# B&R Automation Studio project NAEUL004C00R13L518F00 (part 62)

#### Local.var
```iecst
(*2020-09-10*)
(**)
(*Local Action, State & Status*)
VAR
	eAct : eHermesAction := HermesActIdle;
	eStat : eHermesAction := HermesActIdle;
	eMainStatus : eFBStatus := Idle;
	eStatus : eFBStatus := Idle;
	eStatus1 : eFBStatus := Idle;
	eStatus2 : eFBStatus := Idle;
	eStatus3 : eFBStatus := Idle;
	eStatus4 : eFBStatus := Idle;
	udiStatus : UDINT := 0;
	udiStatus1 : UDINT := 0;
	udiStatus2 : UDINT := 0;
	udiStatus3 : UDINT := 0;
	udiStatus4 : UDINT := 0;
	udiStatus5 : UDINT := 0;
	sStatTxt : STRING[200] := '';
	a_sStatText : ARRAY[0..50] OF STRING[200] := ['Idling','Background Starting Operations','Background Stopping Operations','Deleting Old Log File','Creating Directory','Writing Retain File','Reading Retain File','Saving Configuration',43('')];
END_VAR
(**)
(*Local Alarm*)
VAR
	tyAlmData : tyAlmDat;
	tyAlmData1 : tyAlmDat;
	tyAlmData2 : tyAlmDat;
	tyAlmData3 : tyAlmDat;
	tyAlmData4 : tyAlmDat;
	tyAlmData5 : tyAlmDat;
	tyInfoData : tyAlmDat;
	tyInfoData1 : tyAlmDat;
	tyInfoData2 : tyAlmDat;
	a_tyAlmText : ARRAY[10000..10199] OF tyAlmTxt := [(sAlmText:='Invalid Ident While Client Connecting',sRcyText:='Problem Occurred In The TCP/IP Connection. Check The Connection And Try To Reconnect.'),(sAlmText:='Setting Keep Alive Interval Time Error While Client Connecting',sRcyText:='Unable To Establish Connection Between Machine. Check For Setting And Resume Operation.'),(sAlmText:='Setting Keep Alive Idle Time Error While Client Connecting',sRcyText:='Unable To Establish Connection Between Machine. Check For Setting And Resume Operation.'),(sAlmText:='Setting Keep Alive Count Error While Client Connecting',sRcyText:='Unable To Establish Connection Between Machine. Check For Setting And Resume Operation.'),(sAlmText:='Setting Keep Alive Error While Client Connecting',sRcyText:='Unable To Establish Connection Between Machine. Check For Setting And Resume Operation.'),(sAlmText:='Setting Receive Buffer Error While Client Connecting',sRcyText:='Unable To Establish Connection Between Machine. Check For Setting And Resume Operation.'),(sAlmText:='Setting Send Buffer Error While Client Connecting',sRcyText:='Unable To Establish Connection Between Machine. Check For Setting And Resume Operation.'),(sAlmText:='Setting No Waiting Error While Client Connecting',sRcyText:='Unable To Establish Connection Between Machine. Check For Setting And Resume Operation.'),(sAlmText:='TCP Open Port Error While Client Connecting',sRcyText:='Problem Occurred In The TCP/IP Connection. Check The Connection And Try To Reconnect.'),(sAlmText:='Closing TCP Error While Client Connecting',sRcyText:='Problem Occurred In The TCP/IP Connection. Check The Connection And Try To Reconnect.'),(sAlmText:='Server Connection Failed While Client Connecting',sRcyText:='There Was A Problem Connecting To The Server. The Server May Not Exist or It is Unavailable At This Time. Check The Connection and Try Again.'),(sAlmText:='Ident In Used While Client Connecting',sRcyText:='Problem Occurred In The TCP/IP Connection. Check The Connection And Reconnect.'),(sAlmText:='Connect To Server Error While Client Connecting',sRcyText:='There Was A Problem Connecting To The Server. The Server May Not Exist or It is Unavailable At This Time. Check The Connection and Try Again.'),(sAlmText:='US Hermes Connection Lost',sRcyText:='Please Check Network Connection.'),(sAlmText:='Invalid Ident While Receiving Data',sRcyText:='Problem Occurred In The TCP/IP Connection. Check The Connection And Try To Reconnect.'),(sAlmText:='TCP Receive Data Error While Receiving Data',sRcyText:='Problem Occurred In The TCP/IP Connection. Check The Connection And Try To Reconnect.'),(sAlmText:='Receive ServiceDescription While Upstream In Not Connected State',sRcyText:='Receive Illegal Message.'),(sAlmText:='Receive BoardAvailable While Upstream In Not Connected State',sRcyText:='Receive Illegal Message.'),(sAlmText:='Receive RevokeBoardAvailable While Upstream In Not Connected State',sRcyText:='Receive Illegal Message.'),(sAlmText:='Receive MachineReady While Upstream In Not Connected State',sRcyText:='Receive Illegal Message.'),(sAlmText:='Receive RevokeMachineReady While Upstream In Not Connected State',sRcyText:='Receive Illegal Message.'),(sAlmText:='Receive StartTransport While Upstream In Not Connected State',sRcyText:='Receive Illegal Message.'),(sAlmText:='Receive StopTransport While Upstream In Not Connected State',sRcyText:='Receive Illegal Message.'),(sAlmText:='Receive TransportFinished While Upstream In Not Connected State',sRcyText:='Receive Illegal Message.'),(sAlmText:='Receive BoardForecast While Upstream In Not Connected State',sRcyText:='Receive Illegal Message.'),(sAlmText:='Receive BoardAvailable While Upstream In Service Description State',sRcyText:='Receive Illegal Message.'),(sAlmText:='Receive RevokeBoardAvailable While Upstream In Service Description State',sRcyText:='Receive Illegal Message.'),(sAlmText:='Receive MachineReady While Upstream In Service Description State',sRcyText:='Receive Illegal Message.'),(sAlmText:='Receive RevokeMachineReady While Upstream In Service Description State',sRcyText:='Receive Illegal Message.'),(sAlmText:='Receive StartTransport While Upstream In Service Description State',sRcyText:='Receive Illegal Message.'),(sAlmText:='Receive StopTransport While Upstream In Service Description State',sRcyText:='Receive Illegal Message.'),(sAlmText:='Receive TransportFinished While Upstream In Service Description State',sRcyText:='Receive Illegal Message.'),(sAlmText:='Receive BoardForecast While Upstream In Service Description State',sRcyText:='Receive Illegal Message.'),(sAlmText:='Receive ServiceDescription While Upstream In Not Available Not Ready State',sRcyText:='Receive Illegal Message.'),(sAlmText:='Receive RevokeBoardAvailable While Upstream In Not Available Not Ready State',sRcyText:='Receive Illegal Message.'),(sAlmText:='Receive MachineReady While Upstream In Not Available Not Ready State',sRcyText:='Receive Illegal Message.'),(sAlmText:='Receive RevokeMachineReady While Upstream In Not Available Not Ready State',sRcyText:='Receive Illegal Message.'),(sAlmText:='Receive StartTransport While Upstream In Not Available Not Ready State',sRcyText:='Receive Illegal Message.'),(sAlmText:='Receive StopTransport While Upstream In Not Available Not Ready State',sRcyText:='Receive Illegal Message.'),(sAlmText:='Receive TransportFinished While Upstream In Not Available Not Ready State',sRcyText:='Receive Illegal Message.'),(sAlmText:='Receive ServiceDescription While Upstream In Board Available State',sRcyText:='Receive Illegal Message.'),(sAlmText:='Receive BoardAvailable While Upstream In Board Available State',sRcyText:='Receive Illegal Message.'),(sAlmText:='Receive MachineReady While Upstream In Board Available State',sRcyText:='Receive Illegal Message.'),(sAlmText:='Receive RevokeMachineReady While Upstream In Board Available State',sRcyText:='Receive Illegal Message.'),(sAlmText:='Receive StartTransport While Upstream In Board Available State',sRcyText:='Receive Illegal Message.'),(sAlmText:='Receive StopTransport While Upstream In Board Available State',sRcyText:='Receive Illegal Message.'),(sAlmText:='Receive TransportFinished While Upstream In Board Available State',sRcyText:='Receive Illegal Message.'),(sAlmText:='Receive BoardForecast While Upstream In Board Available State',sRcyText:='Receive Illegal Message.'),(sAlmText:='Receive ServiceDescription While Upstream In Machine Ready State',sRcyText:='Receive Illegal Message.'),(sAlmText:='Receive RevokeBoardAvailable While Upstream In Machine Ready State',sRcyText:='Receive Illegal Message.'),(sAlmText:='Receive MachineReady While Upstream In Machine Ready State',sRcyText:='Receive Illegal Message.'),(sAlmText:='Receive RevokeMachineReady While Upstream In Machine Ready State',sRcyText:='Receive Illegal Message.'),(sAlmText:='Receive StartTransport While Upstream In Machine Ready State',sRcyText:='Receive Illegal Message.'),(sAlmText:='Receive StopTransport While Upstream In Machine Ready State',sRcyText:='Receive Illegal Message.'),(sAlmText:='Receive TransportFinished While Upstream In Machine Ready State',sRcyText:='Receive Illegal Message.'),(sAlmText:='Receive ServiceDescription While Upstream In Available And Ready State',sRcyText:='Receive Illegal Message.'),(sAlmText:='Receive BoardAvailable While Upstream In Available And Ready State',sRcyText:='Receive Illegal Message.'),(sAlmText:='Receive MachineReady While Upstream In Available And Ready State',sRcyText:='Receive Illegal Message.'),(sAlmText:='Receive RevokeMachineReady While Upstream In Available And Ready State',sRcyText:='Receive Illegal Message.'),(sAlmText:='Receive StartTransport While Upstream In Available And Ready State',sRcyText:='Receive Illegal Message.'),(sAlmText:='Receive StopTransport While Upstream In Available And Ready State',sRcyText:='Receive Illegal Message.'),(sAlmText:='Receive TransportFinished While Upstream In Available And Ready State',sRcyText:='Receive Illegal Message.'),(sAlmText:='Receive BoardForecast While Upstream In Available And Ready State',sRcyText:='Receive Illegal Message.'),(sAlmText:='Receive ServiceDescription While Upstream In Transporting State',sRcyText:='Receive Illegal Message.'),(sAlmText:='Receive Twice Board Available While Upstream In Transporting State',sRcyText:='Receive Illegal Message.'),(sAlmText:='Receive RevokeBoardAvailable Without BoardAvailable While Upstream In Transporting State',sRcyText:='Receive Illegal Message.'),(sAlmText:='Receive MachineReady While Upstream In Transporting State',sRcyText:='Receive Illegal Message.'),(sAlmText:='Receive RevokeMachineReady While Upstream In Transporting State',sRcyText:='Receive Illegal Message.'),(sAlmText:='Receive StartTransport While Upstream In Transporting State',sRcyText:='Receive Illegal Message.'),(sAlmText:='Receive StopTransport While Upstream In Transporting State',sRcyText:='Receive Illegal Message.'),(sAlmText:='Receive ServiceDescription While Upstream In Transport Finished State',sRcyText:='Receive Illegal Message.'),(sAlmText:='Receive BoardAvailable While Upstream In Transport Finished State',sRcyText:='Receive Illegal Message.'),(sAlmText:='Receive RevokeBoardAvailable While UpstreamWhile Upstream In Transport Finished State',sRcyText:='Receive Illegal Message.'),(sAlmText:='Receive MachineReady While Upstream In Transport Finished State',sRcyText:='Receive Illegal Message.'),(sAlmText:='Receive RevokeMachineReady While Upstream In Transport Finished State',sRcyText:='Receive Illegal Message.'),(sAlmText:='Receive StartTransport While Upstream In Transport Finished State',sRcyText:='Receive Illegal Message.'),(sAlmText:='Receive TransportFinished While Upstream In Transport Finished State',sRcyText:='Receive Illegal Message.'),(sAlmText:='Receive StopTransport While Upstream In Transport Finished State',sRcyText:='Receive Illegal Message.'),(sAlmText:='Receive BoardForecast While Upstream In Transport Finished State',sRcyText:='Receive Illegal Message.'),(sAlmText:='Receive ServiceDescription While Upstream In Transport Stopped State',sRcyText:='Receive Illegal Message.'),(sAlmText:='Receive Twice Board Available While Upstream In Transport Stopped State',sRcyText:='Receive Illegal Message.'),(sAlmText:='Receive RevokeBoardAvailable Without BoardAvailable While Upstream In Transport Stopped State',sRcyText:='Receive Illegal Message.'),(sAlmText:='Receive MachineReady While Upstream In Transport Stopped State',sRcyText:='Receive Illegal Message.'),(sAlmText:='Receive RevokeMachineReady While Upstream In Transport Stopped State',sRcyText:='Receive Illegal Message.'),(sAlmText:='Receive StartTransport While Upstream In Transport Stopped State',sRcyText:='Receive Illegal Message.'),(sAlmText:='Receive StopTransport While Upstream In Transport Stopped State',sRcyText:='Receive Illegal Message.'),(sAlmText:='LaneId Mismatch While Checking Service Description',sRcyText:='The LaneId Value Does Not Match. Change The Value And Resend The Value.'),(sAlmText:='MachineId Missing While Checking Service Description',sRcyText:='Missing Input Value For MachineId. Fill Up The Value And Resend.'),(sAlmText:='LandId Out Of Range While Checking Service Description',sRcyText:='LaneId Does Not Fall Within The Expected Range.'),(sAlmText:='LandId Missing While Checking Service Description',sRcyText:='Missing Input Value For LaneId. Fill Up The Value And Resend.'),(sAlmText:='Version Missing While Checking Service Description',sRcyText:='Missing Input Value For Version. Fill Up The Value And Resend.'),(sAlmText:='SupportedFeatures Missing While Checking Service Description',sRcyText:='Missing Input Value For SupportedFeatures. Fill Up The Value And Resend.'),(sAlmText:='NotificationCode Out Of Range While Checking Notification',sRcyText:='NotificationCode Does Not Fall Within The Expected Range.'),(sAlmText:='NotificationCode Missing While Checking Notification',sRcyText:='Missing Input Value For NotificationCode. Fill Up The Value And Resend.'),(sAlmText:='Severity Missing While Checking Notification',sRcyText:='Missing Input Value For Severity. Fill Up The Value And Resend.'),(sAlmText:='Description Missing While Checking Notification',sRcyText:='Missing Input Value For Description. Fill Up The Value And Resend.'),(sAlmText:='BoardId Missing While Checking Board Available',sRcyText:='Missing Input Value For BoardId. Fill Up The Value And Resend.'),(sAlmText:='BoardIdCreatedBy Missing While Checking Board Available',sRcyText:='Missing Input Value For BoardIdCreatedBy. Fill Up The Value And Resend.'),(sAlmText:='FailedBoard Missing While Checking Board Available',sRcyText:='Missing Input Value For FailedBoard. Fill Up The Value And Resend.'),(sAlmText:='FlippedBoard Missing While Checking Board Available',sRcyText:='Missing Input Value For FlippedBoard. Fill Up The Value And Resend.'),(sAlmText:='TransferState Missing While Checking Transport Finished',sRcyText:='Missing Input Value For TransferState. Fill Up The Value And Resend.'),(sAlmText:='BoardId Missing While Checking Transport Finished',sRcyText:='Missing Input Value For BoardId. Fill Up The Value And Resend.'),(sAlmText:='FailedBoard Missing While Checking Board Forecast',sRcyText:='Missing Input Value For FailedBoard. Fill Up The Value And Resend.'),(sAlmText:='FlippedBoard Missing While Checking Board Forecast',sRcyText:='Missing Input Value For FlippedBoard. Fill Up The Value And Resend.'),(sAlmText:='BoardId Mismatch While Checking Start Transport & Transport Finished',sRcyText:='The BoardId Value Does Not Match. Change The Value And Resend The Value.'),(sAlmText:='BoardId Missing While Checking Start Transport & Transport Finished',sRcyText:='Missing Input Value For BoardId. Fill Up The Value And Resend.'),(sAlmText:='Service Description Interchange Time Out',sRcyText:='Timeout Expired Before Operation Completed. Reset And Resume Operation.'),(sAlmText:='Transport Time Out',sRcyText:='Timeout Expired Before Operation Completed. Reset And Resume Operation.'),(sAlmText:='Input First Slot Is Invalid',sRcyText:='Invalid Input Value.'),(sAlmText:='Input Last Slot Is Invalid',sRcyText:='Invalid Input Value.'),(sAlmText:='Input Pitch Is Invalid',sRcyText:='Invalid Input Value.'),(sAlmText:='Input Slot To Slot Distance Is Invalid',sRcyText:='Invalid Input Value.'),(sAlmText:='Input Total Slot Is Invalid',sRcyText:='Invalid Input Value.'),(sAlmText:='Input Thickness Is Invalid',sRcyText:='Invalid Input Value.'),(sAlmText:='Input Top Clearance Height Is Invalid',sRcyText:='Invalid Input Value.'),(sAlmText:='Input Bottom Clearance Height Is Invalid',sRcyText:='Invalid Input Value.'),(sAlmText:='Recipe First Slot Value & Board Available Data Not Match With Same Product Type Id',sRcyText:='The Recipe First Slot Value & Board Available Data Value Does Not Match With Product Type ID. Change The Value And Resend The Value.'),(sAlmText:='Recipe Last Slot Value & Board Available Data Not Match With Same Product Type Id',sRcyText:='The Recipe Last Slot Value & Board Available Data Value Does Not Match With Product Type ID. Change The Value And Resend The Value.'),(sAlmText:='Recipe Pitch Value & Board Available Data Not Match With Same Product Type Id',sRcyText:='The Recipe Pitch Value & Board Available Data Value Does Not Match With Product Type ID. Change The Value And Resend The Value.'),(sAlmText:='Width Different With Same Product Type Id',sRcyText:='Width Does Not Match With Product Type ID. Change The Value And Resend The Value.'),(sAlmText:='Input First Slot Is Invalid',sRcyText:='Invalid Input Value.'),(sAlmText:='Input Last Slot Is Invalid',sRcyText:='Invalid Input Value.'),(sAlmText:='Input Pitch Is Invalid',sRcyText:='Invalid Input Value.'),(sAlmText:='Input Slot To Slot Distance Is Invalid',sRcyText:='Invalid Input Value.'),(sAlmText:='Input Total Slot Is Invalid',sRcyText:='Invalid Input Value.'),(sAlmText:='Input Thickness Is Invalid',sRcyText:='Invalid Input Value.'),(sAlmText:='Input Top Clearance Height Is Invalid',sRcyText:='Invalid Input Value.'),(sAlmText:='Input Bottom Clearance Height Is Invalid',sRcyText:='Invalid Input Value.'),(sAlmText:='Recipe First Slot Value & Board Available Data Not Match With Same Product Type Id',sRcyText:='The Recipe First Slot Value & Board Available Data Value Does Not Match With Product Type ID. Change The Value And Resend The Value.'),(sAlmText:='Recipe Last Slot Value & Board Available Data Not Match With Same Product Type Id',sRcyText:='The Recipe Last Slot Value & Board Available Data Value Does Not Match With Product Type ID. Change The Value And Resend The Value.'),(sAlmText:='Recipe Pitch Value & Board Available Data Not Match With Same Product Type Id',sRcyText:='The Recipe Pitch Value & Board Available Data Value Does Not Match With Product Type ID. Change The Value And Resend The Value.'),(sAlmText:='Width Different With Same Product Type Id',sRcyText:='Width Does Not Match With Product Type ID. Change The Value And Resend The Value.'),(sAlmText:='Check Alive Time Out',sRcyText:='Timeout Expired Before Operation Completed. Reset And Resume Operation.'),(sAlmText:='Waiting Check Alive Time Out',sRcyText:='Timeout Expired Before Operation Completed. Reset And Resume Operation.'),(sAlmText:='Check Alive Id Mismatch',sRcyText:='The Check Alive Id Value Does Not Match. Change The Value And Resend The Value.'),(sAlmText:='Board Available Request To Send From Upstream Hermes',sRcyText:='Sending Illegal Message.'),(sAlmText:='Revoke Board Available Request To Send From Upstream Hermes',sRcyText:='Sending Illegal Message.'),(sAlmText:='Transport Finished Request To Send From Upstream Hermes',sRcyText:='Sending Illegal Message.'),(sAlmText:='Set Configuration Request To Send From Upstream Hermes',sRcyText:='Sending Illegal Message.'),(sAlmText:='Get Configuration Request To Send From Upstream Hermes',sRcyText:='Sending Illegal Message.'),(sAlmText:='Current Configuration Request To Send From Upstream Hermes',sRcyText:='Sending Illegal Message.'),(sAlmText:='Board Forecast Request To Send From Upstream Hermes',sRcyText:='Sending Illegal Message.'),(sAlmText:='Query Board Info Request To Send From Upstream Hermes',sRcyText:='Sending Illegal Message.'),(sAlmText:='Invalid Ident While Sending Data',sRcyText:='Invalid Ident Value.'),(sAlmText:='TCP Retry Send Data Error While Sending Data',sRcyText:='Problem Occurred In The TCP/IP Connection. Check The Connection And Try To Reconnect.'),(sAlmText:='TCP Send Data Error',sRcyText:='Problem Occurred In The TCP/IP Connection. Check The Connection And Try To Reconnect.'),(sAlmText:='Invalid Ident While Closing TCP',sRcyText:='Invalid Ident Value.'),(sAlmText:='Closing TCP Error',sRcyText:='Problem Occurred In The TCP/IP Connection. Check The Connection And Try To Reconnect.'),(sAlmText:='File Open Error While Writing Log',sRcyText:='An Error Was Encountered While Trying To Open File. Please Contact Nutek For A Possible Solution.'),(sAlmText:='File Create Error While Writing Log',sRcyText:='An Error Was Encountered While Trying To Create File. Please Contact Nutek For A Possible Solution.'),(sAlmText:='Get File Info Error While Writing Log',sRcyText:='An Error Was Encountered While Getting File Info. Please Contact Nutek For A Possible Solution.'),(sAlmText:='File Write Error While Writing Log',sRcyText:='An Error Was Encountered While Trying To Write File. Please Contact Nutek For A Possible Solution.'),(sAlmText:='File Close Error While Writing Log',sRcyText:='An Error Was Encountered While Trying To Close File. Please Contact Nutek For A Possible Solution.'),(sAlmText:='Directory Does Not Exist While Writing Log',sRcyText:='The Directory Does Not Exist.Please Contact Nutek For A Possible Solution.'),(sAlmText:='Get Directory Info Error While Deleting Old Log',sRcyText:='An Error Was Encountered While Getting Directory Info. Please Contact Nutek For A Possible Solution.'),(sAlmText:='Directory Read Error While Deleting Old Log',sRcyText:='An Error Was Encountered While Reading Directory. Please Contact Nutek For A Possible Solution.'),(sAlmText:='File Delete Error While Deleting Old Log',sRcyText:='An Error Was Encountered While Trying To Delete File. Please Contact Nutek For A Possible Solution.'),(sAlmText:='Board Jam At Sensor After Transfer Interrupted',sRcyText:='Push Back Board To Upstream Machine'),(sAlmText:='Product Type Id Not Receive From Upstream',sRcyText:='Check Upstream Machine Whether Product Type Id Is Used.'),(sAlmText:='Send Board Info Request To Send From Upstream Hermes',sRcyText:='Sending Illegal Message.'),(sAlmText:='Query Work Order Info Request To Send From Upstream Hermes',sRcyText:='Sending Illegal Message.'),(sAlmText:='Send Work Order Info Request To Send From Upstream Hermes',sRcyText:='Sending Illegal Message.'),(sAlmText:='Board Arrived Request To Send From Upstream Hermes',sRcyText:='Sending Illegal Message.'),(sAlmText:='Board Departed Request To Send From Upstream Hermes',sRcyText:='Sending Illegal Message.'),5((0)),(sAlmText:='New Recipe Not Found In Product Recipe List',sRcyText:='Create New Recipe In Product Setting.'),(sAlmText:='Top Barcode Mismatch While Checking SendBoardInfo & QueryBoardInfo',sRcyText:='Wrong Board Info Received. Pleae Check Again.'),(sAlmText:='Top Barcode Missing While Checking SendBoardInfo & QueryBoardInfo',sRcyText:='Wrong Board Info Received. Pleae Check Again.'),(sAlmText:='Bottom Barcode Mismatch While Checking SendBoardInfo & QueryBoardInfo',sRcyText:='Wrong Board Info Received. Pleae Check Again.'),(sAlmText:='Bottom Barcode Missing While Checking SendBoardInfo & QueryBoardInfo',sRcyText:='Wrong Board Info Received. Pleae Check Again.'),26((0))];
END_VAR
(**)
(*Local Output*)
VAR
	a_tyXMLTableDataBrdAvl : ARRAY[0..200] OF tyXMLTableDat;
	iXMLTableDataBrdAvlTtlIdx : INT;
	bConnected : BOOL;
	bHandshakeDone : BOOL;
	bAccDataReq : BOOL;
	bBFAccDataReq : BOOL;
	bOverWriteSlt : BOOL;
	bOverWriteWidth : BOOL;
	bBFOverWriteSlt : BOOL;
	bBFOverWriteWidth : BOOL;
	sReqRecipeNm : STRING[254];
	diReqWidthInUM : DINT;
	diReqMinSltValue : DINT;
	diReqMaxSltValue : DINT;
	diReqPitch : DINT;
	bNotAvlNotRdy : BOOL;
	bBoardAvailable : BOOL;
	bUSRdy : BOOL;
	bDSRdy : BOOL;
	bUSGdRdy : BOOL;
	bDSGdRdy : BOOL;
	bTransporting : BOOL;
	bStopTransport : BOOL;
	bBlkUS2 : BOOL;
	sInternalSnd : STRING[65535];
	bAccDataMnl : BOOL;
	bBFAccDataMnl : BOOL;
	bStopTransportSnd : BOOL;
	tyBoardArrivedInfo : tyHermesBoardAvailable;
	bRcvBoardInfoOk : BOOL;
	bRcvBoardInfoIncompl : BOOL;
	tySendBoardInfoAcc : tyHermesSendBoardInfo;
	tNextPCBTm : TIME;
	bBfReceivedInRdyState : BOOL;
	bBaReceivedInRdyState : BOOL;
END_VAR
(**)
(*Local Input*)
VAR
	udiRstErr : UDINT := 0;
	bPrep : BOOL := TRUE;
	bEn : BOOL := TRUE;
	bDis : BOOL := FALSE;
	tyParam : tyHermesUSParam := (tSndAlive:=T#30s,tRcvAlive:=T#60s,iLaneID:=1,sHostAddress:='192.168.0.200',uiHostPort:=5000);
	sIPAddr : STRING[15] := '192.168.0.100';
	tyDTStructure : DTStructure := (year:=2020,month:=11,day:=11,wday:=05,hour:=21,minute:=28,second:=30,millisec:=123,microsec:=456);
	dtCurrDT : DATE_AND_TIME := DT#2019-02-23-12:30:50;
	bRdyRcv : BOOL := FALSE;
	bRdyTransport : BOOL := FALSE;
	bRcvCompl : BOOL := FALSE;
	bRcvInCompl : BOOL := FALSE;
	bRcvNotStart : BOOL := FALSE;
	bBAWidthEn : BOOL := TRUE; (*Board Available Check Width*)
	bBASltEn : BOOL := FALSE; (*Board Available Check Slot*)
	bBFWidthEn : BOOL := TRUE; (*Board Forecast Check Width*)
	bBFSltEn : BOOL := FALSE; (*Board Forecast Check Slot*)
	sMcId : STRING[80] := '';
	sInterfaceId : STRING[80] := '';
	sVersion : STRING[7] := '1.3';
	eFailedBoard : eHermesFailedBoard := HermesUnknownBoard;
	sRecipeNm : STRING[254] := '';
	diWidthInUM : DINT := 0;
	diMinSltValue : DINT := 0;
	diMaxSltValue : DINT := 0;
	diPitch : DINT := 0;
	diTtlSlt : DINT := 0;
	diSltToSltInUM : DINT := 0;
	udiSndBffrSize : UDINT := 65536;
	udiRcvBffrSize : UDINT := 65536;
	udiAliveIdleTimeInSec : UDINT := 5;
	tConnTimeOut : TIME := T#30s;
	diTransferInTO : DINT := 30000;
	bOpsRun : BOOL := FALSE;
	bInterruptSen : BOOL := FALSE;
	udiFileKeepDay : UDINT := 30;
	sProgNm : STRING[15] := 'USHermes';
	bNtSettingsLoadDone : BOOL := TRUE;
	bAccDataRdy : BOOL := FALSE;
	bRmtPrep : BOOL := FALSE;
	bRmtEn : BOOL := FALSE;
	bSvyPrep : BOOL := FALSE;
	bSvyEn : BOOL := FALSE;
	bAccNewRcpCond : BOOL;
	sInfoMsg : STRING[200] := '';
	sInfoMsg1 : STRING[200] := '';
	sInfoMsg2 : STRING[200] := '';
	a_tyProdRcpList : ARRAY[1..c_udiProdRcpMax] OF tyProdRcpParam;
	tyProdRcpCurrRcp : tyProdRcpParam;
	bMcParamMnlAccData : BOOL;
	bUIAccData : BOOL;
	bQueryBoardInfo : BOOL;
	sTopBarcode : STRING[254] := '';
	sBottomBarcode : STRING[254] := '';
	bInternalUse : BOOL;
	sInternalRcv : STRING[65535];
	tyHermesCurrConfiguration : tyHermesConfiguration;
	bTransportFinished : BOOL;
	bManualInsertEndSen : BOOL;
	bManualInsertZoneHvBrd : BOOL;
	bOpsGConv1HvBrd : BOOL;
	bBAAccpt : BOOL;
	bBFAccpt : BOOL;
END_VAR
(**)
(*Local*)
VAR
	bRstErr : BOOL;
	udiRstErrOld : UDINT;
	bInitDone : BOOL;
	bInitialDone : BOOL;
	bRun : BOOL;
	bStop : BOOL;
	bRstConnection : BOOL;
	bRstState : BOOL;
	udiTCPIdent : UDINT;
	udiXMLTableWriteIdx : UDINT;
	udiMsgSendBffr : UDINT;
	udiSndMsgLen : UDINT;
	sSnd : STRING[65535];
	sRcv : STRING[65535];
	a_tyXMLTableDataRcv : ARRAY[0..200] OF tyXMLTableDat;
	a_tyXMLTableDataSnd : ARRAY[0..200] OF tyXMLTableDat;
	a_eMsgSend : ARRAY[0..50] OF eHermesMsgType;
	tyMsgTypeRcv : tyHermesMsgType;
	tyCheckAliveSnd : tyHermesCheckAlive;
	tyCheckAlivePingSnd : tyHermesCheckAlive;
	tyCheckAlivePongSnd : tyHermesCheckAlive;
	tyCheckAliveRcv : tyHermesCheckAlive;
	tyCheckAlivePingRcv : tyHermesCheckAlive;
	tyCheckAlivePongRcv : tyHermesCheckAlive;
	tyServiceDescriptionSnd : tyHermesServiceDescription;
	tyServiceDescriptionRcv : tyHermesServiceDescription;
	tyNotificationSnd : tyHermesNotification;
	tyNotificationRcv : tyHermesNotification;
	tyBoardAvailableRcv : tyHermesBoardAvailable;
	tyMachineReady : tyHermesMachineReady;
	tyStartTransport : tyHermesStartTransport;
	tyStopTransport : tyHermesStopTransport;
	tyTransportFinished : tyHermesTransportFinished;
	tySetConfiguration : tyHermesSetConfiguration;
	tyCurrentConfiguration : tyHermesCurrentConfiguration;
	tyBoardForecastAcc : tyHermesBoardForecast;
	tyBoardForecastRcv : tyHermesBoardForecast;
	tyQueryBoardInfo : tyHermesQueryBoardInfo;
	tySendBoardInfoRcv : tyHermesSendBoardInfo;
	fbClntConnect : fbTCPClntConnect;
	fbRcv : fbTCPRcv;
	fbSend : fbTCPSnd;
	fbClose : fbTCPClose;
	fbParseXMLTable : fbHermesParseXMLTable;
	fbCheckAlive : fbHermesCheckAlive;
	fbCheckAliveSendPing : fbHermesCheckAliveSendPing;
	fbCheckAliveRcvPing : fbHermesCheckAliveRcvPing;
	fbSequenceUS : fbHermesSequenceUS;
	fbSequenceTO : fbHermesSequenceTO;
	fbGetSlt : fbHermesGetSlt;
	eStatOld : eHermesAction := HermesActIdle;
	tyParamOld : tyHermesUSParam;
	bBlkUS : BOOL;
	bBABlkUS : BOOL;
	bBFBlkUS : BOOL;
	bManuallInsertLastZone : BOOL;
	udiLogCntr : UDINT := 1;
	udiWriteLogCntr : UDINT := 1;
	a_sLogList : ARRAY[1..10] OF STRING[65535];
	sDT : STRING[80];
	dtCurrDTTemp : DATE_AND_TIME;
	fbFileAppend1 : fbFileFullAppend;
	fbFileOldDel1 : fbFileOldDel;
	iWriteLogStep : INT := 0;
	i : INT;
	usiBFAccDataStep : USINT;
	usiAccDataStep : USINT;
	bFeatureBoardForecast : BOOL;
	bProcessBoardForecastId : BOOL;
	fbSendTm : TON;
	fbCheckBATimer : TON;
	fbDelayTm : TON;
	fbUSBlkTm : TON := (PT:=T#1s);
	bReplyMcRdyId : BOOL;
	fbDlyTmr : TON := (PT:=T#5s);
	fbDeleteLogTmr : TON := (PT:=T#24h);
	sTopBtmBarcode : ARRAY[0..1] OF STRING[254];
	udiModuleNum : UDINT := 3101;
END_VAR
```

#### Act_Alarm2.st
```iecst
(** 2019-03-25 **)
ACTION Act_Alarm2:

	//Error
	IF EDGEPOS(eStatus2 = Error) THEN

		tyAlmData2.sProgNm		:= p_sProgNm;
		tyAlmData2.udiCode		:= udiStatus2;
		tyAlmData2.eSeverity	:= AlmSeverityError;
		tyAlmData2.udiRunTime	:= tyAlmData2.udiRunTime + 1;
		tyAlmData2.bAlm			:= TRUE;
		tyAlmData2.udiModuleNum  := udiModuleNum;
		g_sUSHermesAProgNm		:= p_sProgNm;
		//Get Error Message
		IF tyAlmData2.udiCode < 10000 OR tyAlmData2.udiCode > 10199 THEN
			tyAlmData2.sAlmMsg	:= 'Unknown';
			tyAlmData2.sRcyMsg	:= 'Unknown';
		ELSE
			tyAlmData2.sAlmMsg	:= a_tyAlmText[tyAlmData2.udiCode].sAlmText;
			tyAlmData2.sRcyMsg	:= a_tyAlmText[tyAlmData2.udiCode].sRcyText;
		END_IF

		sStatTxt	:= tyAlmData2.sAlmMsg;

	ELSIF bRstErr AND (tyAlmData2.udiCode <> 0) THEN

		tyAlmData2.udiCode		:= 0;
		tyAlmData2.eSeverity	:= AlmSeverityNA;
		tyAlmData2.sAlmMsg		:= '';
		tyAlmData2.sRcyMsg		:= '';
		tyAlmData2.bAlm			:= FALSE;
		sStatTxt	:= a_sStatText[eStat];

	END_IF

END_ACTION
```

#### Act_Alarm4.st
```iecst
(** 2019-03-25 **)
ACTION Act_Alarm4:

	//Error
	IF EDGEPOS(eStatus4 = Error) THEN

		tyAlmData4.sProgNm		:= p_sProgNm;
		tyAlmData4.udiCode		:= udiStatus4;
		tyAlmData4.eSeverity	:= AlmSeverityError;
		tyAlmData4.udiRunTime	:= tyAlmData4.udiRunTime + 1;
		tyAlmData4.bAlm			:= TRUE;
		tyAlmData4.udiModuleNum  := udiModuleNum;
		g_sUSHermesAProgNm		:= p_sProgNm;
		//Get Error Message
		IF tyAlmData4.udiCode < 10000 OR tyAlmData4.udiCode > 10199 THEN
			tyAlmData4.sAlmMsg	:= 'Unknown';
			tyAlmData4.sRcyMsg	:= 'Unknown';
		ELSE
			tyAlmData4.sAlmMsg	:= a_tyAlmText[tyAlmData4.udiCode].sAlmText;
			tyAlmData4.sRcyMsg	:= a_tyAlmText[tyAlmData4.udiCode].sRcyText;
		END_IF

		sStatTxt	:= tyAlmData4.sAlmMsg;

	ELSIF bRstErr AND (tyAlmData4.udiCode <> 0) THEN

		tyAlmData4.udiCode		:= 0;
		tyAlmData4.eSeverity	:= AlmSeverityNA;
		tyAlmData4.sAlmMsg		:= '';
		tyAlmData4.sRcyMsg		:= '';
		tyAlmData4.bAlm			:= FALSE;
		sStatTxt	:= a_sStatText[eStat];

	END_IF

END_ACTION
```

#### Act_Alarm5.st
```iecst
(** 2020-09-10 **)
ACTION Act_Alarm5:

	//Error
	IF ((bConnected = FALSE) AND (p_eLinkMcParamUSCommMod= McSetCommModHermes)) THEN

		tyAlmData5.sProgNm		:= p_sProgNm;
		tyAlmData5.udiCode		:= udiStatus5;
		tyAlmData5.eSeverity	:= AlmSeverityWarning;
		tyAlmData5.udiRunTime	:= tyAlmData5.udiRunTime + 1;
		tyAlmData5.bWarning			:= TRUE;
		tyAlmData5.udiModuleNum  := udiModuleNum;
		g_sUSHermesAProgNm		:= p_sProgNm;
		//Get Error Message
		IF tyAlmData5.udiCode < 10000 OR tyAlmData5.udiCode > 10199 THEN
			tyAlmData5.sAlmMsg	:= 'Unknown';
			tyAlmData5.sRcyMsg	:= 'Unknown';
		ELSE
			tyAlmData5.sAlmMsg	:= a_tyAlmText[tyAlmData5.udiCode].sAlmText;
			tyAlmData5.sRcyMsg	:= a_tyAlmText[tyAlmData5.udiCode].sRcyText;
		END_IF

		sStatTxt	:= tyAlmData5.sAlmMsg;

	ELSIF (bConnected AND (tyAlmData5.udiCode <> 0)) OR (p_eLinkMcParamUSCommMod= McSetCommModSMEMA)  THEN

		tyAlmData5.udiCode		:= 0;
		tyAlmData5.eSeverity	:= AlmSeverityNA;
		tyAlmData5.sAlmMsg		:= '';
		tyAlmData5.sRcyMsg		:= '';
		tyAlmData5.bWarning			:= FALSE;
		sStatTxt	:= a_sStatText[eStat];

	END_IF

END_ACTION
```

#### Act_Background.st
```iecst
(** 2021-08-01 **)
ACTION Act_Background:

	IF bRun = TRUE THEN
		IF udiTCPIdent = 0 THEN
			IF p_bInternalUse = FALSE THEN
				Act_Background_TCPConnect;

				tyParamOld	:= p_tyParam;
			ELSE
				udiTCPIdent	:= 1;
			END_IF

		ELSE
			IF bRstConnection = FALSE THEN
				Act_Background_TCPRcv;

				Act_Background_NotificationRcv;
				Act_Background_IllegalMsg;
				Act_Background_ChkParamRcv;
				Act_Background_CmpParamRcv;

				IF bHandshakeDone = TRUE THEN
					IF (p_tyParam.tSndAlive <> T#0s) AND (p_tyParam.tRcvAlive <> T#0s) THEN
						IF tyServiceDescriptionRcv.tyData.tySupportedFeatures.bFeatureCheckAliveResponse = TRUE AND p_tyParam.bFeatureCheckAliveResponse = TRUE THEN
							Act_Background_ChkAliveSendPing;
							Act_Background_ChkAliveRcvPing;
						ELSE
							Act_Background_ChkAlive;
						END_IF
					ELSE
						fbCheckAlive(bEn := FALSE);
						fbCheckAliveSendPing(bEn := FALSE);
						fbCheckAliveRcvPing(bEn := FALSE);
					END_IF
				END_IF

				Act_Background_BoardAvailableChk;
				Act_Background_BoardForecastIdChk;
				Act_Background_Sequence;
				Act_Background_SequenceTO;
				Act_Background_Err;

				IF tyServiceDescriptionRcv.tyAvl.tySupportedFeatures.bFeatureSendBoardInfo = TRUE AND p_tyParam.bFeatureQueryBoardInfo AND bHandshakeDone THEN
					Act_Background_QueryBoardInfo;
				END_IF

				Act_Background_ChgConfig;

				Act_Background_TCPSend;

			//	Act_Background_Log;

			ELSE
				Act_Background_TCPClose;

			END_IF

		END_IF

	    Act_Background_Stop;

	END_IF
	Act_Background_Log;

	IF EDGENEG(bRun) OR EDGENEG(udiTCPIdent = 0) THEN
		//Reset
		fbClntConnect(bEn := FALSE);

		bConnected	:= bRun;
	END_IF

	IF EDGENEG(bRun) OR EDGENEG(udiTCPIdent <> 0) THEN
		fbRcv(bEn := FALSE);
		fbSequenceUS(bEn := FALSE);
		fbSequenceTO(bEn := FALSE);
		fbCheckAlive(bEn := FALSE);
		fbCheckAliveSendPing(bEn := FALSE);
		fbCheckAliveRcvPing(bEn := FALSE);
		fbSend(bEn := FALSE);
		fbClose(bEn := FALSE);

//		fbFileAppend1(bEn := FALSE);
//		iWriteLogStep	:= 0;

		bConnected		    := FALSE;
		bHandshakeDone	    := FALSE;
		bBlkUS			    := FALSE;
		bBABlkUS			:= FALSE;
		bBFBlkUS			:= FALSE;
		bManuallInsertLastZone	:= FALSE;
		bAccDataReq		    := FALSE;
		bBFAccDataReq	    := FALSE;
		bOverWriteSlt    	:= FALSE;
		bOverWriteWidth	    := FALSE;
		bBFOverWriteSlt	    := FALSE;
		bBFOverWriteWidth	:= FALSE;
		bRstConnection    	:= FALSE;
		bRstState	    	:= FALSE;
		bUSRdy	    		:= FALSE;
		bDSRdy		    	:= FALSE;
		bTransporting    	:= FALSE;
		bStopTransport   	:= FALSE;

		memset(ADR(tyMsgTypeRcv) , 0 , SIZEOF(tyMsgTypeRcv));
		memset(ADR(a_eMsgSend) , 0 , SIZEOF(a_eMsgSend));
		udiMsgSendBffr	:= 0;
	END_IF

	//Reset Error
	IF (eStatus1 = Error) AND bRstErr THEN
		eStatus1	:= Idle;
		udiStatus1	:= 0;

		fbClntConnect(bEn := FALSE);
		fbRcv(bEn := FALSE);
		fbSequenceUS(bEn := FALSE);
		fbSend(bEn := FALSE);
		fbClose(bEn := FALSE);
		fbCheckAlive(bEn := FALSE);
		fbCheckAliveSendPing(bEn := FALSE);
		fbCheckAliveRcvPing(bEn := FALSE);
		fbSequenceTO(bEn := FALSE);

//		fbFileAppend1(bEn := FALSE);
//		iWriteLogStep	:= 0;

		bConnected		    := FALSE;
		bHandshakeDone	    := FALSE;
		bBlkUS			    := FALSE;
		bBABlkUS			:= FALSE;
		bBFBlkUS			:= FALSE;
		bManuallInsertLastZone	:= FALSE;
		bAccDataReq		    := FALSE;
		bBFAccDataReq	    := FALSE;
		bOverWriteSlt    	:= FALSE;
		bOverWriteWidth	    := FALSE;
		bBFOverWriteSlt	    := FALSE;
		bBFOverWriteWidth	:= FALSE;
		bRstConnection    	:= FALSE;
		bRstState	    	:= FALSE;
		bUSRdy	    		:= FALSE;
		bDSRdy		    	:= FALSE;
		bTransporting    	:= FALSE;
		bStopTransport   	:= FALSE;

		memset(ADR(tyMsgTypeRcv) , 0 , SIZEOF(tyMsgTypeRcv));
		memset(ADR(a_eMsgSend) , 0 , SIZEOF(a_eMsgSend));
		udiMsgSendBffr	:= 0;
	END_IF

	IF (eStatus2 = Error) AND bRstErr THEN
		eStatus2	:= Idle;
		udiStatus2	:= 0;

		fbSequenceTO(bEn := FALSE);

	END_IF

	IF (eStatus3 = Error) AND bRstErr THEN
		eStatus3	:= Idle;
		udiStatus3	:= 0;

//		fbFileAppend1(bEn := FALSE);
//		iWriteLogStep	:= 0;
	END_IF

	IF (eStatus4 = Error) AND bRstErr THEN
		eStatus4	:= Idle;
		udiStatus4	:= 0;
	END_IF

	Act_Background_AccData;
	Act_Background_BFAccData;

END_ACTION
```

#### Act_Background_AccData.st
```iecst
(** 2021-08-01 **)
ACTION Act_Background_AccData: //Accept BoardAvailable Data from Upstream

	CASE usiAccDataStep OF
		0:
			//Request Accept Data
			IF bUSRdy = TRUE AND eMainStatus <> Error AND bAccDataReq = TRUE THEN
				usiAccDataStep	:= 1;
			END_IF
			//bUSRdy := fbSequenceUS.bUSRdy;
			//bUSRdy:= (eState = HermesStateBoardAvailable) OR (eState = HermesStateAvailableAndReady) OR (eState >= HermesStateTransporting);
		1:
			//Manual Accept Data Check
			IF bAccDataReq = TRUE THEN
				IF p_bMcParamMnlAccData = TRUE THEN
					bAccDataMnl	:= TRUE;

					tyInfoData.sProgNm		:= p_sProgNm;
					tyInfoData.udiCode		:= 10000;
					tyInfoData.eSeverity	:= AlmSeverityInfo;
					tyInfoData.sAlmMsg		:= p_sInfoMsg;

					IF p_bUIAccData = TRUE THEN
						p_bUIAccData    := FALSE; //2023_07_26_Debug for Manual Accept Data automatically accept after product change many times
						bAccDataMnl		:= FALSE;
						usiAccDataStep	:= 2;
					END_IF
				ELSE
					bAccDataMnl		:= FALSE;
					p_bUIAccData    := FALSE; //2023_07_26_Debug for Manual Accept Data automatically accept after product change many times
					usiAccDataStep	:= 2;
				END_IF
			ELSE
				bAccDataMnl		:= FALSE;
				usiAccDataStep	:= 4;
			END_IF

		2:
			IF bAccDataReq = TRUE  THEN
				IF p_bAccNewRcpCond = TRUE THEN //In Auto Mode, and empty
					usiAccDataStep	:= 3;
					IF p_bNtParamAutoRcpPrep AND NOT(p_bMcParamAutoRcpDis) THEN
						CASE p_eNtParamAutoRcpPrecededBy OF
							PrecededBySelf:
								usiAccDataStep	:= 4;
							PrecededByF1:
								usiAccDataStep	:= 3;
						END_CASE
					END_IF
				ELSE
					//Info Message
					tyInfoData.sProgNm		:= p_sProgNm;
					tyInfoData.udiCode		:= 10000;
					tyInfoData.eSeverity	:= AlmSeverityInfo;
					tyInfoData.sAlmMsg		:= p_sInfoMsg;
				END_IF
			ELSE
				usiAccDataStep	:= 4;
			END_IF

		3:
			//Sync Recipe
			IF bOverWriteWidth = TRUE OR bOverWriteSlt = TRUE THEN

				//Accept New Recipe Width
				IF bOverWriteWidth = TRUE THEN
					p_tyProdRcpCurrRcp.diWidthInUM	:= diReqWidthInUM;
				END_IF

				//Accept New Recipe Slot
				IF bOverWriteSlt = TRUE THEN
					p_tyProdRcpCurrRcp.diMaxSltValue := diReqMaxSltValue;
					p_tyProdRcpCurrRcp.diMinSltValue := diReqMinSltValue;
					p_tyProdRcpCurrRcp.diPitch		 := diReqPitch;
				END_IF

			ELSE

				//Accept New Recipe Name
				FOR i := 1 TO 2000 DO
					IF sReqRecipeNm = pa_tyProdRcpList[i].sRcpNm THEN
						p_tyProdRcpCurrRcp	:= pa_tyProdRcpList[i];
						EXIT;
					END_IF
				END_FOR

				IF i > 2000 THEN
					//Recipe Not Exist
					eStatus4	:= Error;
					udiStatus4	:= 10169;	//New Recipe Not Found In Product Recipe List

					fHermesAddOneMsgSend(ADR(a_eMsgSend) , ADR(udiMsgSendBffr) , HermesMsgTypeNotification);

					tyNotificationSnd.tyAvl.bSeverity			:= TRUE;
					tyNotificationSnd.tyAvl.bNotificationCode	:= TRUE;
					tyNotificationSnd.tyAvl.bDescription		:= TRUE;
					tyNotificationSnd.tyData.eSeverity			:= HermesSeverityError;
					tyNotificationSnd.tyData.iNotificationCode	:= UDINT_TO_INT(udiStatus4);
					tyNotificationSnd.tyData.sDescription		:= a_tyAlmText[udiStatus4].sAlmText;

				END_IF

			END_IF

			usiAccDataStep	:= 4;

		4:
			//Clear Info Message
			tyInfoData.sProgNm		:= '';
			tyInfoData.udiCode		:= 0;
			tyInfoData.eSeverity	:= AlmSeverityNA;
			tyInfoData.sAlmMsg		:= '';

			usiAccDataStep	:= 0;

	END_CASE

END_ACTION
```

#### Act_Background_BoardAvailableChk.st
```iecst
(** 2021-08-01 **)
ACTION Act_Background_BoardAvailableChk:

	IF eStatus2 <> Error THEN
		     //Add
		//IF p_bNewIncomingBoard = FALSE AND p_bSiemensMcModeChgPrep = FALSE AND
		IF p_bAccDataRdy AND (bTransporting = FALSE) AND(p_bOpsRun = TRUE) THEN
			bBaReceivedInRdyState	:= p_bAccDataRdy AND (bTransporting = FALSE) AND(p_bOpsRun = TRUE);//AutoRcp
			bAccDataReq		:= FALSE;
			bBABlkUS		:= FALSE;
			bOverWriteSlt	:= FALSE;
			bOverWriteWidth	:= FALSE;

			IF p_tyParam.bCmpTypeId = TRUE  THEN	//"Compare Type ID" Ticked

				IF tyBoardAvailableRcv.tyAvl.bProductTypeId = TRUE THEN	//Check if there is Product Type Id in B.A msg

					IF tyBoardAvailableRcv.tyData.sProductTypeId <> p_sRecipeNm THEN	//Product Type Id Different

						bAccDataReq	    := TRUE;	//Require To Load New Recipe
						bBABlkUS		:= TRUE;

						sReqRecipeNm	:= tyBoardAvailableRcv.tyData.sProductTypeId;
						diReqWidthInUM	:= REAL_TO_DINT(tyBoardAvailableRcv.tyData.rWidth * 1000);

					ELSE	//Product Type Id Same (After accepted or Originally same)

						IF p_tyParam.bCmpParam = TRUE THEN	//"Compare Param" Ticked
							IF tyBoardAvailableRcv.tyAvl.bThickness AND tyBoardAvailableRcv.tyAvl.bTopClearanceHeight AND tyBoardAvailableRcv.tyAvl.bBottomClearanceHeight AND p_bBASltEn THEN	//Camparing Slot Parameters if p_bBASltEn = TRUE
								udiStatus2	:= fHermesCmpSlt(tyBoardAvailableRcv.tyData.eFlippedBoard , tyBoardAvailableRcv.tyData.rThickness , tyBoardAvailableRcv.tyData.rTopClearanceHeight , tyBoardAvailableRcv.tyData.rBottomClearanceHeight , p_diMinSltValue , p_diMaxSltValue , p_diPitch , p_diSltToSltInUM , p_diTtlSlt);

								IF udiStatus2 <> 0 THEN

									bBABlkUS	:= TRUE;

									eStatus2	:= Error;

									IF udiStatus2 = 2914 THEN
										udiStatus2	:= 10108;	//Input First Slot Is Invalid
									ELSIF udiStatus2 = 2915 THEN
										udiStatus2	:= 10109;	//Input Last Slot Is Invalid
									ELSIF udiStatus2 = 2916 THEN
										udiStatus2	:= 10110;	//Input Pitch Is Invalid
									ELSIF udiStatus2 = 2917 THEN
										udiStatus2	:= 10111;	//Input Slot To Slot Distance Is Invalid
									ELSIF udiStatus2 = 2918 THEN
										udiStatus2	:= 10112;	//Input Total Slot Is Invalid
									ELSIF udiStatus2 = 2919 THEN
										udiStatus2	:= 10113;	//Input Thickness Is Invalid
									ELSIF udiStatus2 = 2920 THEN
										udiStatus2	:= 10114;	//Input Top Clearance Height Is Invalid
									ELSIF udiStatus2 = 2921 THEN
										udiStatus2	:= 10115;	//Input Bottom Clearance Height Is Invalid
									ELSIF udiStatus2 = 2922 THEN
										udiStatus2	:= 10116;	//Recipe First Slot Value & Board Available Data Not Match With Same Product Type Id
									ELSIF udiStatus2 = 2923 THEN
										udiStatus2	:= 10117;	//Recipe Last Slot Value & Board Available Data Not Match With Same Product Type Id
									ELSIF udiStatus2 = 2924 THEN
										udiStatus2	:= 10118;	//Recipe Pitch Value & Board Available Data Not Match With Same Product Type Id
									END_IF

									fHermesAddOneMsgSend(ADR(a_eMsgSend) , ADR(udiMsgSendBffr) , HermesMsgTypeNotification);

									tyNotificationSnd.tyAvl.bSeverity			:= TRUE;
									tyNotificationSnd.tyAvl.bNotificationCode	:= TRUE;
									tyNotificationSnd.tyAvl.bDescription		:= TRUE;
									tyNotificationSnd.tyData.eSeverity			:= HermesSeverityError;
									tyNotificationSnd.tyData.iNotificationCode	:= UDINT_TO_INT(udiStatus2);
									tyNotificationSnd.tyData.sDescription		:= a_tyAlmText[udiStatus2].sAlmText;

								END_IF
							END_IF

							IF tyBoardAvailableRcv.tyAvl.bWidth AND p_bBAWidthEn THEN	//Comparing Width Parameter if p_bBAWidthEn = TRUE
								IF REAL_TO_DINT(tyBoardAvailableRcv.tyData.rWidth * 1000) <> p_diWidthInUM THEN

									bBABlkUS	:= TRUE;

									eStatus2	:= Error;
									udiStatus2	:= 10119;	//Width Different With Same Product Type Id

									fHermesAddOneMsgSend(ADR(a_eMsgSend) , ADR(udiMsgSendBffr) , HermesMsgTypeNotification);

									tyNotificationSnd.tyAvl.bSeverity			:= TRUE;
									tyNotificationSnd.tyAvl.bNotificationCode	:= TRUE;
									tyNotificationSnd.tyAvl.bDescription		:= TRUE;
									tyNotificationSnd.tyData.eSeverity			:= HermesSeverityError;
									tyNotificationSnd.tyData.iNotificationCode	:= UDINT_TO_INT(udiStatus2);
									tyNotificationSnd.tyData.sDescription		:= a_tyAlmText[udiStatus2].sAlmText;

								END_IF
							END_IF

						END_IF

					END_IF

				ELSE

					eStatus2	:= Error;
					udiStatus2	:= 10158;	//Product Type Id Not Receive From Upstream

					fHermesAddOneMsgSend(ADR(a_eMsgSend) , ADR(udiMsgSendBffr) , HermesMsgTypeNotification);

					tyNotificationSnd.tyAvl.bSeverity			:= TRUE;
					tyNotificationSnd.tyAvl.bNotificationCode	:= TRUE;
					tyNotificationSnd.tyAvl.bDescription		:= TRUE;
					tyNotificationSnd.tyData.eSeverity			:= HermesSeverityError;
					tyNotificationSnd.tyData.iNotificationCode	:= UDINT_TO_INT(udiStatus2);
					tyNotificationSnd.tyData.sDescription		:= a_tyAlmText[udiStatus2].sAlmText;

				END_IF

			ELSE	//"Compare Type ID" Not Ticked
				                                    //Add
				IF p_tyParam.bOverwrite THEN //AND p_bNewIncomingBoard = FALSE  THEN	//"Overwrite" Ticked

					IF tyBoardAvailableRcv.tyAvl.bThickness AND tyBoardAvailableRcv.tyAvl.bTopClearanceHeight AND tyBoardAvailableRcv.tyAvl.bBottomClearanceHeight AND p_bBASltEn THEN	//Camparing Slot Parameters

						udiStatus2	:= fHermesCmpSlt(tyBoardAvailableRcv.tyData.eFlippedBoard , tyBoardAvailableRcv.tyData.rThickness , tyBoardAvailableRcv.tyData.rTopClearanceHeight , tyBoardAvailableRcv.tyData.rBottomClearanceHeight , p_diMinSltValue , p_diMaxSltValue , p_diPitch , p_diSltToSltInUM , p_diTtlSlt);

						IF udiStatus2 <> 0 THEN

							bAccDataReq		:= TRUE;
							bBABlkUS			:= TRUE;
							bOverWriteSlt	:= TRUE;

							fbGetSlt.eFlippedBrd				:= tyBoardAvailableRcv.tyData.eFlippedBoard;
							fbGetSlt.rThicknessInMM				:= tyBoardAvailableRcv.tyData.rThickness;
							fbGetSlt.rTopClearanceHeightInMM	:= tyBoardAvailableRcv.tyData.rTopClearanceHeight;
							fbGetSlt.rBtmClearanceHeightInMM	:= tyBoardAvailableRcv.tyData.rBottomClearanceHeight;
							fbGetSlt.diSltToSltInUM				:= p_diSltToSltInUM;
							fbGetSlt.diTtlSlt					:= p_diTtlSlt;
							fbGetSlt;

							diReqMinSltValue	:= fbGetSlt.diMinSltValue;
							diReqMaxSltValue	:= fbGetSlt.diMaxSltValue;
							diReqPitch			:= fbGetSlt.diPitch;

						END_IF

					END_IF

					IF tyBoardAvailableRcv.tyAvl.bWidth  AND p_bBAWidthEn THEN // AND p_usiLinkProdRcpCurrRcpMcMod = 0 THEN	//Comparing Width Parameter
						IF REAL_TO_DINT(tyBoardAvailableRcv.tyData.rWidth * 1000) <> p_diWidthInUM THEN

							bAccDataReq		:= TRUE;
							bBABlkUS		:= TRUE;
							bOverWriteWidth	:= TRUE;

							diReqWidthInUM	:= REAL_TO_DINT(tyBoardAvailableRcv.tyData.rWidth * 1000);

						END_IF
					END_IF

				ELSE	//"Compare Type ID" Not Ticked and "Overwrite" Not Ticked, Error if not same

					IF tyBoardAvailableRcv.tyAvl.bThickness AND tyBoardAvailableRcv.tyAvl.bTopClearanceHeight AND tyBoardAvailableRcv.tyAvl.bBottomClearanceHeight AND p_bBASltEn AND p_bRdyRcv THEN	//Camparing Slot Parameters
						udiStatus2	:= fHermesCmpSlt(tyBoardAvailableRcv.tyData.eFlippedBoard , tyBoardAvailableRcv.tyData.rThickness , tyBoardAvailableRcv.tyData.rTopClearanceHeight , tyBoardAvailableRcv.tyData.rBottomClearanceHeight , p_diMinSltValue , p_diMaxSltValue , p_diPitch , p_diSltToSltInUM , p_diTtlSlt);

						IF udiStatus2 <> 0 THEN

							bBABlkUS		:= TRUE;

							eStatus2	:= Error;

							IF udiStatus2 = 2914 THEN
								udiStatus2	:= 10120;	//Input First Slot Is Invalid
							ELSIF udiStatus2 = 2915 THEN
								udiStatus2	:= 10121;	//Input Last Slot Is Invalid
							ELSIF udiStatus2 = 2916 THEN
								udiStatus2	:= 10122;	//Input Pitch Is Invalid
							ELSIF udiStatus2 = 2917 THEN
								udiStatus2	:= 10123;	//Input Slot To Slot Distance Is Invalid
							ELSIF udiStatus2 = 2918 THEN
								udiStatus2	:= 10124;	//Input Total Slot Is Invalid
							ELSIF udiStatus2 = 2919 THEN
								udiStatus2	:= 10125;	//Input Thickness Is Invalid
							ELSIF udiStatus2 = 2920 THEN
								udiStatus2	:= 10126;	//Input Top Clearance Height Is Invalid
							ELSIF udiStatus2 = 2921 THEN
								udiStatus2	:= 10127;	//Input Bottom Clearance Height Is Invalid
							ELSIF udiStatus2 = 2922 THEN
								udiStatus2	:= 10128;	//Recipe First Slot Value & Board Available Data Not Match With Same Product Type Id
							ELSIF udiStatus2 = 2923 THEN
								udiStatus2	:= 10129;	//Recipe Last Slot Value & Board Available Data Not Match With Same Product Type Id
							ELSIF udiStatus2 = 2924 THEN
								udiStatus2	:= 10130;	//Recipe Pitch Value & Board Available Data Not Match With Same Product Type Id
							END_IF

							fHermesAddOneMsgSend(ADR(a_eMsgSend) , ADR(udiMsgSendBffr) , HermesMsgTypeNotification);

							tyNotificationSnd.tyAvl.bSeverity			:= TRUE;
							tyNotificationSnd.tyAvl.bNotificationCode	:= TRUE;
							tyNotificationSnd.tyAvl.bDescription		:= TRUE;
							tyNotificationSnd.tyData.eSeverity			:= HermesSeverityError;
							tyNotificationSnd.tyData.iNotificationCode	:= UDINT_TO_INT(udiStatus2);
							tyNotificationSnd.tyData.sDescription		:= a_tyAlmText[udiStatus2].sAlmText;

						END_IF
					END_IF

					IF tyBoardAvailableRcv.tyAvl.bWidth AND p_bBAWidthEn AND p_bRdyRcv THEN	//Comparing Width Parameter
						IF REAL_TO_DINT(tyBoardAvailableRcv.tyData.rWidth * 1000) <> p_diWidthInUM THEN

							bBABlkUS		:= TRUE;

							eStatus2	:= Error;
							udiStatus2	:= 10131;	//Width Different With Same Product Type Id

							fHermesAddOneMsgSend(ADR(a_eMsgSend) , ADR(udiMsgSendBffr) , HermesMsgTypeNotification);

							tyNotificationSnd.tyAvl.bSeverity			:= TRUE;
							tyNotificationSnd.tyAvl.bNotificationCode	:= TRUE;
							tyNotificationSnd.tyAvl.bDescription		:= TRUE;
							tyNotificationSnd.tyData.eSeverity			:= HermesSeverityError;
							tyNotificationSnd.tyData.iNotificationCode	:= UDINT_TO_INT(udiStatus2);
							tyNotificationSnd.tyData.sDescription		:= a_tyAlmText[udiStatus2].sAlmText;

						END_IF
					END_IF

				END_IF

			END_IF

		ELSIF (p_bAccDataRdy = FALSE) OR bTransporting = TRUE THEN
			bBaReceivedInRdyState	:= FALSE;//AutoRcp
			bAccDataReq		:= FALSE;
			bBABlkUS		:= FALSE;
			bOverWriteSlt	:= FALSE;
			bOverWriteWidth	:= FALSE;
			sTopBtmBarcode[0] := tyBoardAvailableRcv.tyData.sTopBarcode;
			sTopBtmBarcode[1] := tyBoardAvailableRcv.tyData.sBottomBarcode;

		END_IF

	ELSE

		bAccDataReq		:= FALSE;
		bBABlkUS		:= TRUE;
		bOverWriteSlt	:= FALSE;
		bOverWriteWidth	:= FALSE;
		sTopBtmBarcode[0] 	:= '';
		sTopBtmBarcode[1] 	:= '';

		bBaReceivedInRdyState := FALSE; //AutoRcp
	END_IF

END_ACTION
```

#### Act_Background_BoardForecastIdChk.st
```iecst
(** 2021-08-01 **)
ACTION Act_Background_BoardForecastIdChk:

	IF eStatus2 <> Error  THEN

		IF bProcessBoardForecastId AND bNotAvlNotRdy AND (bTransporting = FALSE) AND (p_bOpsRun = TRUE) AND p_bSiemensMcModeChgPrep = FALSE THEN
			bBfReceivedInRdyState := 	bProcessBoardForecastId AND bNotAvlNotRdy AND (bTransporting = FALSE) AND (p_bOpsRun = TRUE)  ;	 //AutoRcp
			bBFAccDataReq		:= FALSE;
			bBFBlkUS			:= FALSE;
			bBFOverWriteSlt  	:= FALSE;
			bBFOverWriteWidth	:= FALSE;
			                                      //Add
			IF p_tyParam.bCmpTypeId = TRUE THEN // AND p_bNewIncomingBoard = FALSE  THEN	//"Compare Type ID" Ticked

				IF tyBoardForecastAcc.tyAvl.bProductTypeId = TRUE THEN	//Check if there is Product Type Id in B.F msg

					IF tyBoardForecastAcc.tyData.sProductTypeId <> p_sRecipeNm THEN	//Product Type Id Different

						bBFAccDataReq	:= TRUE;	//Require To Load New Recipe
						bBFBlkUS		:= TRUE;

						sReqRecipeNm	:= tyBoardForecastAcc.tyData.sProductTypeId;
						diReqWidthInUM	:= REAL_TO_DINT(tyBoardForecastAcc.tyData.rWidth * 1000);

					ELSE	//Product Type Id Same (After accepted or Originally same)

						IF p_tyParam.bCmpParam = TRUE THEN	//"Compare Param" Ticked
							IF tyBoardForecastAcc.tyAvl.bThickness AND tyBoardForecastAcc.tyAvl.bTopClearanceHeight AND tyBoardForecastAcc.tyAvl.bBottomClearanceHeight AND p_bBFSltEn THEN	//Camparing Slot Parameters if p_bBFSltEn = TRUE
								udiStatus2	:= fHermesCmpSlt(tyBoardForecastAcc.tyData.eFlippedBoard , tyBoardForecastAcc.tyData.rThickness , tyBoardForecastAcc.tyData.rTopClearanceHeight , tyBoardForecastAcc.tyData.rBottomClearanceHeight , p_diMinSltValue , p_diMaxSltValue , p_diPitch , p_diSltToSltInUM , p_diTtlSlt);

								IF udiStatus2 <> 0 THEN

									bBFBlkUS		:= TRUE;
									bProcessBoardForecastId := FALSE;//add
									eStatus2	:= Error;

									IF udiStatus2 = 2914 THEN
										udiStatus2	:= 10108;	//Input First Slot Is Invalid
									ELSIF udiStatus2 = 2915 THEN
										udiStatus2	:= 10109;	//Input Last Slot Is Invalid
									ELSIF udiStatus2 = 2916 THEN
										udiStatus2	:= 10110;	//Input Pitch Is Invalid
									ELSIF udiStatus2 = 2917 THEN
										udiStatus2	:= 10111;	//Input Slot To Slot Distance Is Invalid
									ELSIF udiStatus2 = 2918 THEN
										udiStatus2	:= 10112;	//Input Total Slot Is Invalid
									ELSIF udiStatus2 = 2919 THEN
										udiStatus2	:= 10113;	//Input Thickness Is Invalid
									ELSIF udiStatus2 = 2920 THEN
										udiStatus2	:= 10114;	//Input Top Clearance Height Is Invalid
									ELSIF udiStatus2 = 2921 THEN
										udiStatus2	:= 10115;	//Input Bottom Clearance Height Is Invalid
									ELSIF udiStatus2 = 2922 THEN
										udiStatus2	:= 10116;	//Recipe First Slot Value & Board Available Data Not Match With Same Product Type Id
									ELSIF udiStatus2 = 2923 THEN
										udiStatus2	:= 10117;	//Recipe Last Slot Value & Board Available Data Not Match With Same Product Type Id
									ELSIF udiStatus2 = 2924 THEN
										udiStatus2	:= 10118;	//Recipe Pitch Value & Board Available Data Not Match With Same Product Type Id
									END_IF

									fHermesAddOneMsgSend(ADR(a_eMsgSend) , ADR(udiMsgSendBffr) , HermesMsgTypeNotification);

									tyNotificationSnd.tyAvl.bSeverity			:= TRUE;
									tyNotificationSnd.tyAvl.bNotificationCode	:= TRUE;
									tyNotificationSnd.tyAvl.bDescription		:= TRUE;
									tyNotificationSnd.tyData.eSeverity			:= HermesSeverityError;
									tyNotificationSnd.tyData.iNotificationCode	:= 6; //BoardForecast Error
									tyNotificationSnd.tyData.sDescription		:= a_tyAlmText[udiStatus2].sAlmText;

								END_IF
							END_IF

							IF tyBoardForecastAcc.tyAvl.bWidth AND p_bBFWidthEn THEN	//Comparing Width Parameter if p_bBFWidthEn = TRUE
								IF REAL_TO_DINT(tyBoardForecastAcc.tyData.rWidth * 1000) <> p_diWidthInUM THEN

									bBFBlkUS	:= TRUE;
									bProcessBoardForecastId := FALSE;//add
									eStatus2	:= Error;
									udiStatus2	:= 10119;	//Width Different With Same Product Type Id

									fHermesAddOneMsgSend(ADR(a_eMsgSend) , ADR(udiMsgSendBffr) , HermesMsgTypeNotification);

									tyNotificationSnd.tyAvl.bSeverity			:= TRUE;
									tyNotificationSnd.tyAvl.bNotificationCode	:= TRUE;
									tyNotificationSnd.tyAvl.bDescription		:= TRUE;
									tyNotificationSnd.tyData.eSeverity			:= HermesSeverityError;
									tyNotificationSnd.tyData.iNotificationCode	:= 6; //BoardForecast Error
									tyNotificationSnd.tyData.sDescription		:= a_tyAlmText[udiStatus2].sAlmText;
								ELSE
									bReplyMcRdyId           := TRUE; //add
									bProcessBoardForecastId := FALSE; //add
								END_IF
							END_IF

						END_IF

					END_IF

				ELSE

					eStatus2	:= Error;
					udiStatus2	:= 10158;	//Product Type Id Not Receive From Upstream
					bProcessBoardForecastId := FALSE;//add

					fHermesAddOneMsgSend(ADR(a_eMsgSend) , ADR(udiMsgSendBffr) , HermesMsgTypeNotification);

					tyNotificationSnd.tyAvl.bSeverity			:= TRUE;
					tyNotificationSnd.tyAvl.bNotificationCode	:= TRUE;
					tyNotificationSnd.tyAvl.bDescription		:= TRUE;
					tyNotificationSnd.tyData.eSeverity			:= HermesSeverityError;
					tyNotificationSnd.tyData.iNotificationCode	:= 6; //BoardForecast Error
					tyNotificationSnd.tyData.sDescription		:= a_tyAlmText[udiStatus2].sAlmText;

				END_IF

			ELSE	//"Compare Type ID" Not Ticked

				IF p_tyParam.bOverwrite THEN // AND p_bNewIncomingBoard = FALSE   THEN	//"Overwrite" Ticked

					IF tyBoardForecastAcc.tyAvl.bThickness AND tyBoardForecastAcc.tyAvl.bTopClearanceHeight AND tyBoardForecastAcc.tyAvl.bBottomClearanceHeight AND p_bBFSltEn THEN	//Camparing Slot Parameters

						udiStatus2	:= fHermesCmpSlt(tyBoardForecastAcc.tyData.eFlippedBoard , tyBoardForecastAcc.tyData.rThickness , tyBoardForecastAcc.tyData.rTopClearanceHeight , tyBoardForecastAcc.tyData.rBottomClearanceHeight , p_diMinSltValue , p_diMaxSltValue , p_diPitch , p_diSltToSltInUM , p_diTtlSlt);

						IF udiStatus2 <> 0 THEN

							bBFAccDataReq		:= TRUE;
							bBFBlkUS			:= TRUE;
							bBFOverWriteSlt	    := TRUE;

							fbGetSlt.eFlippedBrd				:= tyBoardForecastAcc.tyData.eFlippedBoard;
							fbGetSlt.rThicknessInMM				:= tyBoardForecastAcc.tyData.rThickness;
							fbGetSlt.rTopClearanceHeightInMM	:= tyBoardForecastAcc.tyData.rTopClearanceHeight;
							fbGetSlt.rBtmClearanceHeightInMM	:= tyBoardForecastAcc.tyData.rBottomClearanceHeight;
							fbGetSlt.diSltToSltInUM				:= p_diSltToSltInUM;
							fbGetSlt.diTtlSlt					:= p_diTtlSlt;
							fbGetSlt;

							diReqMinSltValue	:= fbGetSlt.diMinSltValue;
							diReqMaxSltValue	:= fbGetSlt.diMaxSltValue;
							diReqPitch			:= fbGetSlt.diPitch;

						END_IF

					END_IF

					IF tyBoardForecastAcc.tyAvl.bWidth AND p_bBFWidthEn THEN	//Comparing Width Parameter
						IF REAL_TO_DINT(tyBoardForecastAcc.tyData.rWidth * 1000) <> p_diWidthInUM THEN

							bBFAccDataReq		:= TRUE;
							bBFBlkUS			:= TRUE;
							bBFOverWriteWidth	:= TRUE;

							diReqWidthInUM	:= REAL_TO_DINT(tyBoardForecastAcc.tyData.rWidth * 1000);
						ELSE
							bReplyMcRdyId           := TRUE; //add
							bProcessBoardForecastId := FALSE; //add
						END_IF
					END_IF

				ELSE	//"Compare Type ID" Not Ticked and "Overwrite" Not Ticked, Error if not same

					IF tyBoardForecastAcc.tyAvl.bThickness AND tyBoardForecastAcc.tyAvl.bTopClearanceHeight AND tyBoardForecastAcc.tyAvl.bBottomClearanceHeight AND p_bBFSltEn AND p_bRdyRcv THEN	//Camparing Slot Parameters
						udiStatus2	:= fHermesCmpSlt(tyBoardForecastAcc.tyData.eFlippedBoard , tyBoardForecastAcc.tyData.rThickness , tyBoardForecastAcc.tyData.rTopClearanceHeight , tyBoardForecastAcc.tyData.rBottomClearanceHeight , p_diMinSltValue , p_diMaxSltValue , p_diPitch , p_diSltToSltInUM , p_diTtlSlt);

						IF udiStatus2 <> 0 THEN

							bBFBlkUS		:= TRUE;
							bProcessBoardForecastId := FALSE;//add
							eStatus2	:= Error;

							IF udiStatus2 = 2914 THEN
								udiStatus2	:= 10120;	//Input First Slot Is Invalid
							ELSIF udiStatus2 = 2915 THEN
								udiStatus2	:= 10121;	//Input Last Slot Is Invalid
							ELSIF udiStatus2 = 2916 THEN
								udiStatus2	:= 10122;	//Input Pitch Is Invalid
							ELSIF udiStatus2 = 2917 THEN
								udiStatus2	:= 10123;	//Input Slot To Slot Distance Is Invalid
							ELSIF udiStatus2 = 2918 THEN
								udiStatus2	:= 10124;	//Input Total Slot Is Invalid
							ELSIF udiStatus2 = 2919 THEN
								udiStatus2	:= 10125;	//Input Thickness Is Invalid
							ELSIF udiStatus2 = 2920 THEN
								udiStatus2	:= 10126;	//Input Top Clearance Height Is Invalid
							ELSIF udiStatus2 = 2921 THEN
								udiStatus2	:= 10127;	//Input Bottom Clearance Height Is Invalid
							ELSIF udiStatus2 = 2922 THEN
								udiStatus2	:= 10128;	//Recipe First Slot Value & Board Available Data Not Match With Same Product Type Id
							ELSIF udiStatus2 = 2923 THEN
								udiStatus2	:= 10129;	//Recipe Last Slot Value & Board Available Data Not Match With Same Product Type Id
							ELSIF udiStatus2 = 2924 THEN
								udiStatus2	:= 10130;	//Recipe Pitch Value & Board Available Data Not Match With Same Product Type Id
							END_IF

							fHermesAddOneMsgSend(ADR(a_eMsgSend) , ADR(udiMsgSendBffr) , HermesMsgTypeNotification);

							tyNotificationSnd.tyAvl.bSeverity			:= TRUE;
							tyNotificationSnd.tyAvl.bNotificationCode	:= TRUE;
							tyNotificationSnd.tyAvl.bDescription		:= TRUE;
							tyNotificationSnd.tyData.eSeverity			:= HermesSeverityError;
							tyNotificationSnd.tyData.iNotificationCode	:= 6; //BoardForecast Error
							tyNotificationSnd.tyData.sDescription		:= a_tyAlmText[udiStatus2].sAlmText;

						END_IF
					END_IF

					IF tyBoardForecastAcc.tyAvl.bWidth AND p_bBFWidthEn AND p_bRdyRcv THEN	//Comparing Width Parameter
						IF REAL_TO_DINT(tyBoardForecastAcc.tyData.rWidth * 1000) <> p_diWidthInUM THEN

							bBFBlkUS		:= TRUE;
							bProcessBoardForecastId := FALSE;//add
							eStatus2	:= Error;
							udiStatus2	:= 10131;	//Width Different With Same Product Type Id

							fHermesAddOneMsgSend(ADR(a_eMsgSend) , ADR(udiMsgSendBffr) , HermesMsgTypeNotification);

							tyNotificationSnd.tyAvl.bSeverity			:= TRUE;
							tyNotificationSnd.tyAvl.bNotificationCode	:= TRUE;
							tyNotificationSnd.tyAvl.bDescription		:= TRUE;
							tyNotificationSnd.tyData.eSeverity			:= HermesSeverityError;
							tyNotificationSnd.tyData.iNotificationCode	:= 6; //BoardForecast Error
							tyNotificationSnd.tyData.sDescription		:= a_tyAlmText[udiStatus2].sAlmText;
						ELSE
							bReplyMcRdyId           := TRUE; //add
							bProcessBoardForecastId := FALSE; //add
						END_IF
					END_IF

				END_IF

			END_IF

		ELSIF bProcessBoardForecastId = FALSE OR bNotAvlNotRdy =FALSE OR bTransporting = TRUE THEN
			bBfReceivedInRdyState := 	FALSE;
			bBFAccDataReq		:= FALSE;
			bBFBlkUS			:= FALSE;
			bBFOverWriteSlt	    := FALSE;
			bBFOverWriteWidth	:= FALSE;

		END_IF

	ELSE

		bBFAccDataReq		:= FALSE;
		bBFBlkUS			:= TRUE;
		bBFOverWriteSlt	    := FALSE;
		bBFOverWriteWidth	:= FALSE;

		bBfReceivedInRdyState := FALSE; //AutoRcp
	END_IF

END_ACTION
```

#### Act_Background_ChkAlive.st
```iecst
(** 2021-08-01 **)
ACTION Act_Background_ChkAlive:

	IF eStatus1 <> Error THEN

		//Standard Check Alive (Without Ping & Pong)
		fbCheckAlive.bDataRcv		:= tyMsgTypeRcv.bCheckAlive OR tyMsgTypeRcv.bBoardAvailable OR tyMsgTypeRcv.bRevokeBoardAvailable OR tyMsgTypeRcv.bTransportFinished OR tyMsgTypeRcv.bBoardForecast OR tyMsgTypeRcv.bSendBoardInfo;
		fbCheckAlive.tSendTm		:= p_tyParam.tSndAlive;
		fbCheckAlive.tRcvTimeOut	:= p_tyParam.tRcvAlive;
		fbCheckAlive(bEn := TRUE);

		IF fbCheckAlive.udiStatus > 0 AND fbCheckAlive.udiStatus < 65534 THEN
			eStatus1	:= Error;

			IF fbCheckAlive.udiStatus = 2767 THEN
				udiStatus1	:= 10132;	//Check Alive Time Out
			ELSE
				udiStatus1	:= fbCheckAlive.udiStatus;
			END_IF

			fHermesAddOneMsgSend(ADR(a_eMsgSend) , ADR(udiMsgSendBffr) , HermesMsgTypeNotification);

			tyNotificationSnd.tyAvl.bSeverity			:= TRUE;
			tyNotificationSnd.tyAvl.bNotificationCode	:= TRUE;
			tyNotificationSnd.tyAvl.bDescription		:= TRUE;
			tyNotificationSnd.tyData.eSeverity			:= HermesSeverityFatalError;
			tyNotificationSnd.tyData.iNotificationCode	:= UDINT_TO_INT(udiStatus1);
			tyNotificationSnd.tyData.sDescription		:= a_tyAlmText[udiStatus1].sAlmText;

		ELSE
			IF EDGEPOS(fbCheckAlive.bDataSend) THEN
				fHermesAddOneMsgSend(ADR(a_eMsgSend) , ADR(udiMsgSendBffr) , HermesMsgTypeCheckAlive);
				tyCheckAliveSnd	:= fbCheckAlive.tyDataSend;
			END_IF

		END_IF

		tyMsgTypeRcv.bCheckAlive	:= FALSE;	//Reset Check Alive

	END_IF

END_ACTION
```

#### Act_Background_ChkParamRcv.st
```iecst
(** 2021-08-01 **)
ACTION Act_Background_ChkParamRcv:

	IF eStatus2 <> Error THEN

		//Check Parameter Receive
		IF tyMsgTypeRcv.bServiceDescription = TRUE THEN
			udiStatus2	:= fHermesChkParamSD(tyServiceDescriptionRcv , p_tyParam.iLaneID);

			IF udiStatus2 = 2731 THEN
				udiStatus2	:= 0;
			END_IF

			IF udiStatus2 <> 0 THEN
				eStatus2	:= Error;

				IF udiStatus2 = 2726 THEN
					udiStatus2	:= 10086;	//LaneId Mismatch While Checking Service Description
				ELSIF udiStatus2 = 2727 THEN
					udiStatus2	:= 10087;	//MachineId Missing While Checking Service Description
				ELSIF udiStatus2 = 2728 THEN
					udiStatus2	:= 10088;	//LandId Out Of Range While Checking Service Description
				ELSIF udiStatus2 = 2729 THEN
					udiStatus2	:= 10089;	//LandId Missing While Checking Service Description
				ELSIF udiStatus2 = 2730 THEN
					udiStatus2	:= 10090;	//Version Missing While Checking Service Description
				ELSIF udiStatus2 = 2731 THEN
					udiStatus2	:= 10091;	//SupportedFeatures Missing While Checking Service Description
				END_IF

				fHermesAddOneMsgSend(ADR(a_eMsgSend) , ADR(udiMsgSendBffr) , HermesMsgTypeNotification);

				tyNotificationSnd.tyAvl.bSeverity			:= TRUE;
				tyNotificationSnd.tyAvl.bNotificationCode	:= TRUE;
				tyNotificationSnd.tyAvl.bDescription		:= TRUE;
				tyNotificationSnd.tyData.eSeverity			:= HermesSeverityFatalError;
				tyNotificationSnd.tyData.iNotificationCode	:= UDINT_TO_INT(udiStatus2);
				tyNotificationSnd.tyData.sDescription		:= a_tyAlmText[udiStatus2].sAlmText;

			END_IF
		END_IF

		IF tyMsgTypeRcv.bNotification = TRUE THEN
			udiStatus2	:= fHermesChkParamN(tyNotificationRcv);

			IF udiStatus2 <> 0 THEN
				eStatus2	:= Error;

				IF udiStatus2 = 2732 THEN
					udiStatus2	:= 10092;	//NotificationCode Out Of Range While Checking Notification
				ELSIF udiStatus2 = 2733 THEN
					udiStatus2	:= 10093;	//NotificationCode Missing While Checking Notification
				ELSIF udiStatus2 = 2734 THEN
					udiStatus2	:= 10094;	//Severity Missing While Checking Notification
				ELSIF udiStatus2 = 2735 THEN
					udiStatus2	:= 10095;	//Description Missing While Checking Notification
				END_IF

				fHermesAddOneMsgSend(ADR(a_eMsgSend) , ADR(udiMsgSendBffr) , HermesMsgTypeNotification);

				tyNotificationSnd.tyAvl.bSeverity			:= TRUE;
				tyNotificationSnd.tyAvl.bNotificationCode	:= TRUE;
				tyNotificationSnd.tyAvl.bDescription		:= TRUE;
				tyNotificationSnd.tyData.eSeverity			:= HermesSeverityFatalError;
				tyNotificationSnd.tyData.iNotificationCode	:= UDINT_TO_INT(udiStatus2);
				tyNotificationSnd.tyData.sDescription		:= a_tyAlmText[udiStatus2].sAlmText;

			END_IF
		END_IF

		IF tyMsgTypeRcv.bBoardAvailable = TRUE THEN
			udiStatus2	:= fHermesChkParamBA(tyBoardAvailableRcv);

			IF udiStatus2 <> 0 THEN
				eStatus2	:= Error;

				IF udiStatus2 = 2736 THEN
					udiStatus2	:= 10096;	//BoardId Missing While Checking Board Available
				ELSIF udiStatus2 = 2737 THEN
					udiStatus2	:= 10097;	//BoardIdCreatedBy Missing While Checking Board Available
				ELSIF udiStatus2 = 2738 THEN
					udiStatus2	:= 10098;	//FailedBoard Missing While Checking Board Available
				ELSIF udiStatus2 = 2739 THEN
					udiStatus2	:= 10099;	//FlippedBoard Missing While Checking Board Available
				END_IF

				fHermesAddOneMsgSend(ADR(a_eMsgSend) , ADR(udiMsgSendBffr) , HermesMsgTypeNotification);

				tyNotificationSnd.tyAvl.bSeverity			:= TRUE;
				tyNotificationSnd.tyAvl.bNotificationCode	:= TRUE;
				tyNotificationSnd.tyAvl.bDescription		:= TRUE;
				tyNotificationSnd.tyData.eSeverity			:= HermesSeverityError;
				tyNotificationSnd.tyData.iNotificationCode	:= UDINT_TO_INT(udiStatus2);
				tyNotificationSnd.tyData.sDescription		:= a_tyAlmText[udiStatus2].sAlmText;
//			ELSE
//				IF p_bNtParamAutoRcpPrep AND NOT(p_bMcParamAutoRcpDis) THEN
//					bBAAccpt := TRUE;
//				END_IF
			END_IF
//		ELSE
//			bBAAccpt := FALSE;
		END_IF

		IF tyMsgTypeRcv.bTransportFinished = TRUE THEN
			udiStatus2	:= fHermesChkParamTF(tyTransportFinished);

			IF udiStatus2 <> 0 THEN
				eStatus2	:= Error;

				IF udiStatus2 = 2744 THEN
					udiStatus2	:= 10100;	//TransferState Missing While Checking Transport Finished
				ELSIF udiStatus2 = 2745 THEN
					udiStatus2	:= 10101;	//BoardId Missing While Checking Transport Finished
				END_IF

				fHermesAddOneMsgSend(ADR(a_eMsgSend) , ADR(udiMsgSendBffr) , HermesMsgTypeNotification);

				tyNotificationSnd.tyAvl.bSeverity			:= TRUE;
				tyNotificationSnd.tyAvl.bNotificationCode	:= TRUE;
				tyNotificationSnd.tyAvl.bDescription		:= TRUE;
				tyNotificationSnd.tyData.eSeverity			:= HermesSeverityError;
				tyNotificationSnd.tyData.iNotificationCode	:= UDINT_TO_INT(udiStatus2);
				tyNotificationSnd.tyData.sDescription		:= a_tyAlmText[udiStatus2].sAlmText;

			END_IF
		END_IF

		IF tyMsgTypeRcv.bBoardForecast = TRUE THEN
			IF bFeatureBoardForecast = TRUE THEN

				udiStatus2	:= fHermesChkParamBF(tyBoardForecastRcv);

				IF udiStatus2 <> 0 THEN
					eStatus2	:= Error;

					IF udiStatus2 = 2764 THEN
						udiStatus2	:= 10102;	//FailedBoard Missing While Checking Board Forecast

					ELSIF udiStatus2 = 2765 THEN
						udiStatus2	:= 10103;	//FlippedBoard Missing While Checking Board Forecast
					END_IF

					fHermesAddOneMsgSend(ADR(a_eMsgSend) , ADR(udiMsgSendBffr) , HermesMsgTypeNotification);

					tyNotificationSnd.tyAvl.bSeverity			:= TRUE;
					tyNotificationSnd.tyAvl.bNotificationCode	:= TRUE;
					tyNotificationSnd.tyAvl.bDescription		:= TRUE;
					tyNotificationSnd.tyData.eSeverity			:= HermesSeverityError;
					tyNotificationSnd.tyData.iNotificationCode	:= UDINT_TO_INT(udiStatus2);
					tyNotificationSnd.tyData.sDescription		:= a_tyAlmText[udiStatus2].sAlmText;

				END_IF

			ELSE
				tyMsgTypeRcv.bBoardForecast := FALSE;
			END_IF

		END_IF

	END_IF

END_ACTION
```

#### Act_Background_CmpParamRcv.st
```iecst
(** 2021-08-01 **)
ACTION Act_Background_CmpParamRcv:

	IF eStatus2 <> Error THEN

		IF tyMsgTypeRcv.bTransportFinished = TRUE THEN
			udiStatus2	:= fHermesChkParamSTTF(tyStartTransport , tyTransportFinished);

			IF udiStatus2 <> 0 THEN
				eStatus2	:= Error;

				IF udiStatus2 = 2714 THEN
					udiStatus2	:= 10104;	//BoardId Mismatch While Checking Start Transport & Transport Finished
				ELSIF udiStatus2 = 2715 THEN
					udiStatus2	:= 10105;	//BoardId Missing While Checking Start Transport & Transport Finished
				END_IF

				fHermesAddOneMsgSend(ADR(a_eMsgSend) , ADR(udiMsgSendBffr) , HermesMsgTypeNotification);

				tyNotificationSnd.tyAvl.bSeverity			:= TRUE;
				tyNotificationSnd.tyAvl.bNotificationCode	:= TRUE;
				tyNotificationSnd.tyAvl.bDescription		:= TRUE;
				tyNotificationSnd.tyData.eSeverity			:= HermesSeverityFatalError;
				tyNotificationSnd.tyData.iNotificationCode	:= UDINT_TO_INT(udiStatus2);
				tyNotificationSnd.tyData.sDescription		:= a_tyAlmText[udiStatus2].sAlmText;

			END_IF
		END_IF

		IF tyServiceDescriptionRcv.tyAvl.tySupportedFeatures.bFeatureSendBoardInfo = TRUE AND p_tyParam.bFeatureQueryBoardInfo THEN
			IF tyMsgTypeRcv.bSendBoardInfo = TRUE AND p_bQueryBoardInfo THEN
				udiStatus2	:= fHermesChkParamSBIQBI(tySendBoardInfoRcv , tyQueryBoardInfo);

				IF udiStatus2 <> 0 THEN
					eStatus2	:= Error;

					IF udiStatus2 = 2769 THEN
						udiStatus2	:= 10170;	//Top Barcode Mismatch While Checking SendBoardInfo & QueryBoardInfo
					ELSIF udiStatus2 = 2770 THEN
						udiStatus2	:= 10171;	//Top Barcode Missing While Checking SendBoardInfo & QueryBoardInfo
					ELSIF udiStatus2 = 2771 THEN
						udiStatus2	:= 10172;	//Bottom Barcode Mismatch While Checking SendBoardInfo & QueryBoardInfo
					ELSIF udiStatus2 = 2772 THEN
						udiStatus2	:= 10173;	//Bottom Barcode Missing While Checking SendBoardInfo & QueryBoardInfo
					END_IF

					fHermesAddOneMsgSend(ADR(a_eMsgSend) , ADR(udiMsgSendBffr) , HermesMsgTypeNotification);

					tyNotificationSnd.tyAvl.bSeverity			:= TRUE;
					tyNotificationSnd.tyAvl.bNotificationCode	:= TRUE;
					tyNotificationSnd.tyAvl.bDescription		:= TRUE;
					tyNotificationSnd.tyData.eSeverity			:= HermesSeverityError;
					tyNotificationSnd.tyData.iNotificationCode	:= UDINT_TO_INT(udiStatus2);
					tyNotificationSnd.tyData.sDescription		:= a_tyAlmText[udiStatus2].sAlmText;

					tyMsgTypeRcv.bSendBoardInfo := FALSE; //reset, else will latching
				END_IF
			END_IF
		END_IF

	END_IF

END_ACTION
```

#### Act_Background_NotificationSnd.st
```iecst
(** 2021-08-01 **)
ACTION Act_Background_NotificationSnd:

	IF a_eMsgSend[0] = HermesMsgTypeNotification THEN
		bRstConnection	:= fHermesNotificationRstConn(tyNotificationSnd) OR bRstConnection; //Fatal Error = Reset Connection, Error no reset
//		bRstState		:= fHermesNotificationRstState(tyNotificationSnd) OR bRstState;
	END_IF

END_ACTION
```

#### Act_Background_QueryBoardInfo.st
```iecst
(** 2021-08-01 **)
ACTION Act_Background_QueryBoardInfo:

	IF eStatus2 <> Error THEN

		IF EDGEPOS(p_bQueryBoardInfo) THEN

			fHermesAddOneMsgSend(ADR(a_eMsgSend) , ADR(udiMsgSendBffr) , HermesMsgTypeQueryBoardInfo);

			tyQueryBoardInfo.tyData.sTopBarcode						            := p_sTopBarcode;
			tyQueryBoardInfo.tyData.sBottomBarcode							    := p_sBottomBarcode;

			tyQueryBoardInfo.tyAvl.bTopBarcode									:= tyQueryBoardInfo.tyData.sTopBarcode <> '';
			tyQueryBoardInfo.tyAvl.bBottomBarcode							    := tyQueryBoardInfo.tyData.sBottomBarcode <>'';

		END_IF

		IF tyMsgTypeRcv.bSendBoardInfo THEN

			IF p_bQueryBoardInfo AND (udiStatus2 = 0) THEN //After CmpParamRcv
				IF tySendBoardInfoRcv.tyAvl.bBoardId AND tySendBoardInfoRcv.tyAvl.bBoardIdCreatedBy THEN; // AND p_bManualInsertZoneHvBrd = FALSE AND p_bManualInsertEndSen = FALSE THEN //Wait Empty

					bRcvBoardInfoOk              := TRUE;
					tySendBoardInfoAcc          := tySendBoardInfoRcv;
					tyMsgTypeRcv.bSendBoardInfo := FALSE;

				ELSIF ((tySendBoardInfoRcv.tyAvl.bBoardId = FALSE) OR (tySendBoardInfoRcv.tyAvl.bBoardIdCreatedBy = FALSE)) THEN //no BoardId or BoardIdCreatedBy
					bRcvBoardInfoIncompl := TRUE;
					bManuallInsertLastZone         := FALSE;
					tyMsgTypeRcv.bSendBoardInfo := FALSE;
				END_IF

			ELSIF p_bQueryBoardInfo = FALSE THEN
				tyMsgTypeRcv.bSendBoardInfo     := FALSE;
			END_IF

		END_IF

		IF 	bRcvBoardInfoOk = TRUE THEN
			bManuallInsertLastZone        := TRUE; //Board data received from upstream, block Upstream to allow manual insert

			tyInfoData1.sProgNm		:= p_sProgNm;
			tyInfoData1.udiCode		:= 10000;
			tyInfoData1.eSeverity	:= AlmSeverityInfo;
			tyInfoData1.sAlmMsg		:= p_sInfoMsg1;

			IF p_bTransportFinished THEN

				bRcvBoardInfoOk := FALSE;
				bManuallInsertLastZone        := FALSE;
			END_IF

		ELSIF bRcvBoardInfoIncompl = TRUE THEN //receive dummy, no need block upstream

			tyInfoData2.sProgNm		:= p_sProgNm;
			tyInfoData2.udiCode		:= 10000;
			tyInfoData2.eSeverity	:= AlmSeverityInfo;
			tyInfoData2.sAlmMsg		:= p_sInfoMsg2;

		END_IF

		IF p_bQueryBoardInfo = FALSE THEN

			//Clear Info Message 1
			tyInfoData1.sProgNm		:= '';
			tyInfoData1.udiCode		:= 0;
			tyInfoData1.eSeverity	:= AlmSeverityNA;
			tyInfoData1.sAlmMsg		:= '';
			bRcvBoardInfoOk := FALSE;
			bManuallInsertLastZone        := FALSE;

			//Clear Info Message 2
			tyInfoData2.sProgNm		:= '';
			tyInfoData2.udiCode		:= 0;
			tyInfoData2.eSeverity	:= AlmSeverityNA;
			tyInfoData2.sAlmMsg		:= '';
			bRcvBoardInfoIncompl := FALSE;

		END_IF

	END_IF

END_ACTION
```

#### Act_InitGlobal.st
```iecst
(** 2021-08-01 **)
ACTION Act_InitGlobal:

	(* Always Change If Project Change *)

	//Pass Data To Link
	p_bLinkStartupRun ACCESS p_StartupRun;
	p_eLinkMcParamUSCommMod ACCESS p_McParamUSCommAMod;

	//p_eLinkConvDir ACCESS p_NtParamProjConvDir;
	p_bLinkDILeftSen ACCESS p_DIConvLftSen;
	//p_bLinkDIRightSen ACCESS p_DIConvRgtSen;

	p_eLinkTravLifULPosGo ACCESS p_OpsTravLifULPosGo;
	p_bLinkOpsTravLifULUSComm ACCESS p_OpsTravLifULUSComm;

//	p_bLinkOpsGConv1HvBrd ACCESS p_ConvHvBrd;
//	p_bLinkOpsGConv2HvBrd ACCESS p_OpsGConv2HvBrd; //Zone 2 and so on.
//	p_bLinkOpsGConv1StepChkInitDone ACCESS p_OpsConvStepChkInit;
//	p_bLinkOpsGConv2StepChkInitDone ACCESS p_OpsGConv2StepChkInitDone;  //Zone 2 and so on.
//	p_bLinkDIPresentSen ACCESS p_DIBrdStackPresentSen;

	//Pass Data To Internal Use
	p_udiRstErr ACCESS p_RstErrReset;
	p_bPrep ACCESS p_NtParamHermesPrep;
	p_tyParam ACCESS p_HermesUSParam1;
	p_sIPAddr ACCESS p_HWInfoIPAddr;
	p_tyDTStructure ACCESS p_TimeCurrDTStruct;
	p_dtCurrDT ACCESS p_TimeCurrDT;
	p_sMcId ACCESS p_McParamMcNm;
//	p_sRecipeNm ACCESS p_ProdRcpCurrRcp0Nm;
//	p_diWidthInUM ACCESS p_ProdRcpCurrRcp0Width;
	p_udiAliveIdleTimeInSec ACCESS p_NtParamUSHermesAAliveTmInSec;
	p_tConnTimeOut ACCESS p_NtParamUSHermesAConnTO;
	p_diTransferInTO ACCESS p_McParamTranInErrDlyTm;
	p_bInterruptSen ACCESS p_DIConvLftSen;
	p_bOpsRun ACCESS p_OpsRun;
	p_udiFileKeepDay ACCESS p_NtParamUSHermesAFileKeepDay;
	p_sProgNm ACCESS p_NtParamUSHermesAProgNm;
	p_bNtSettingsLoadDone ACCESS p_StartupNtSettingsLoadDone;
//	p_bAccDataRdy ACCESS p_USHermesUSRdy;
	p_bRmtPrep ACCESS p_NtParamHermesRmtPrep;
	p_bRmtEn ACCESS p_McParamHermesRmtEn;
	p_bSvyPrep ACCESS p_NtParamHermesSvyPrep;
	p_bSvyEn ACCESS p_McParamHermesSvyEn;
	pa_tyProdRcpList ACCESS p_ProdRcpCurrList;
	p_tyProdRcpCurrRcp ACCESS p_ProdRcpCurrRcp0;
	p_bMcParamMnlAccData ACCESS p_McParamMnlAccDat;
	p_bOpsGConv1HvBrd ACCESS p_PshrConvHvBrd;//p_ConvHvBrd; //Take Zone 1's Have Board
	//p_bManualInsertZoneHvBrd ACCESS p_ConvHvBrd; //Take Manual Insesrt Zone's Have Board
	//p_bManualInsertEndSen ACCESS p_DIConvRgtSen; //Manual insert sensor position, for example exit sensor of attached output conveyor, or Last Zone conveyor exit sensor
	p_bUIAccData ACCESS p_UIProdAccData;
	p_bQueryBoardInfo ACCESS p_UIQueryBoardInfo;
	p_sTopBarcode ACCESS p_UITravLifTopBarcode;
	p_sBottomBarcode ACCESS p_UITravLifBottomBarcode;
	p_tyHermesConfiguration ACCESS p_HermesConfiguration;
	//p_bTransportFinished ACCESS p_DSHermesTransportFinishedSnd; //used to reset bManuallInsertLastZone

	p_bSiemensMcModeChgPrep ACCESS p_McParamSiemensPrep;          //ADD   Include ReplyWorkOrderID & Machine mode changeover
	p_usiLinkProdRcpCurrRcpMcMod ACCESS p_ProdRcpCurrRcp0McMod;      //Add
	p_bNewIncomingBoard ACCESS p_NewIncomingBoard;
	p_bQueryBypassWorkOrder ACCESS p_QueryBypassWorkOrder;

	p_bNtParamAutoRcpPrep ACCESS p_NtParamAutoRcpPrep;
	p_bMcParamAutoRcpDis  ACCESS p_McParamAutoRcpDisable;
	p_eNtParamAutoRcpPrecededBy ACCESS p_NtParamAutoRcpPrecededBy;

	(* Always Change If Project Change *)
END_ACTION
```

#### Act_Link.st
```iecst
(** 2019-06-04 **)
ACTION Act_Link:

	//Receive Alive Time
	p_tyParam.tRcvAlive	:= p_tyParam.tSndAlive * 2;

	//Transfer Complete
	p_bRcvCompl	:= EDGENEG(p_bLinkDILeftSen);

	//Ready Receive
	p_bRdyRcv	:= p_bLinkOpsTravLifULUSComm AND p_eLinkTravLifULPosGo = TravLifULPosUS1;

	//Ready Transport
//	p_bRdyTransport	:= TRUE;

	//Accept Data Ready
	IF bUSRdy AND p_eLinkTravLifULPosGo = TravLifULPosUS1 THEN
		p_bAccDataRdy	:= TRUE;
	ELSIF bUSRdy = FALSE THEN
		p_bAccDataRdy	:= FALSE;
	END_IF

	//Accept New Recipe Condition
	p_bAccNewRcpCond	:= p_bOpsRun = TRUE AND p_bOpsGConv1HvBrd = FALSE;

	//Info Message
	p_sInfoMsg		:= 'Upstream Hermes Request New Recipe';
	p_sInfoMsg		:= CONCAT(p_sInfoMsg , '$r$n');
	p_sInfoMsg		:= CONCAT(p_sInfoMsg , 'Old Recipe Name : ');
	p_sInfoMsg		:= CONCAT(p_sInfoMsg , p_sRecipeNm);
	p_sInfoMsg		:= CONCAT(p_sInfoMsg , '$r$n');
	p_sInfoMsg		:= CONCAT(p_sInfoMsg , 'Old Recipe Width : ');
	sWidthInUMTemp	:= DINT_TO_STRING(p_diWidthInUM / 1000);
	p_sInfoMsg		:= CONCAT(p_sInfoMsg , sWidthInUMTemp);
	p_sInfoMsg		:= CONCAT(p_sInfoMsg , '$r$n');
	p_sInfoMsg		:= CONCAT(p_sInfoMsg , 'New Recipe Name : ');
	p_sInfoMsg		:= CONCAT(p_sInfoMsg , sReqRecipeNm);
	p_sInfoMsg		:= CONCAT(p_sInfoMsg , '$r$n');
	p_sInfoMsg		:= CONCAT(p_sInfoMsg , 'New Recipe Width : ');
	sWidthInUMTemp	:= DINT_TO_STRING(diReqWidthInUM / 1000);
	p_sInfoMsg		:= CONCAT(p_sInfoMsg , sWidthInUMTemp);

	//Info Message 1 for "SendBoardInfo"
	p_sInfoMsg1     := 'Board Info Received From Upstream';
	p_sInfoMsg1		:= CONCAT(p_sInfoMsg1 , '$r$n');
	p_sInfoMsg1		:= CONCAT(p_sInfoMsg1 , 'PCB Transfer to Last Zone is Blocked');
	p_sInfoMsg1		:= CONCAT(p_sInfoMsg1 , '$r$n');
	p_sInfoMsg1		:= CONCAT(p_sInfoMsg1 , 'Please Insert PCB to Last Zone Outlet');
	p_sInfoMsg1		:= CONCAT(p_sInfoMsg1 , '$r$n');
	p_sInfoMsg1		:= CONCAT(p_sInfoMsg1 , 'and PCB Data Will Be Overwritten');
	p_sInfoMsg1		:= CONCAT(p_sInfoMsg1 , '$r$n');
	p_sInfoMsg1		:= CONCAT(p_sInfoMsg1 , 'To Cancel,unpress the Query Board Info Button');

	//Info Message 2 for "SendBoardInfo"
	p_sInfoMsg2     := 'Board Info Not Found From Upstream';

	//Block Upstream                                                  //ADD
	//Changed
	bBlkUS :=  bBABlkUS OR bBFBlkUS OR bManuallInsertLastZone; // OR (p_eLinkMcParamUSCommMod = McSetCommModHermes AND (p_bQueryBypassWorkOrder OR p_bNewIncomingBoard)) ; //Remove bManuallInsertLastZone if this is a multiple zones, use bManuallInsertLastZone to block respective zones board transfer

	//bManuallInsertLastZone Waiting Board Transport to DS
	p_bTransportFinished :=  EDGENEG(p_bOpsGConv1HvBrd); // added DSSMEMA if necessary

	//Changed
//	IF p_bNewIncomingBoard = FALSE THEN
//		fbUSBlkTm(IN := TRUE);
//	ELSIF p_bNewIncomingBoard THEN
//		fbUSBlkTm(IN := FALSE);
//	END_IF

	//IF AutoRcp Prep, Link
	IF p_bNtParamAutoRcpPrep AND NOT(p_bMcParamAutoRcpDis) AND p_eNtParamAutoRcpPrecededBy = PrecededBySelf   THEN
		p_sRecipeNm	ACCESS p_AutoRcpCurrRcpProdID;
		p_diWidthInUM ACCESS p_AutoRcpCurrRcpWidth;
	ELSE
		p_sRecipeNm	ACCESS p_ProdRcpCurrRcp0Nm;
		p_diWidthInUM ACCESS p_ProdRcpCurrRcp0Width;
	END_IF

END_ACTION
```

#### Act_LinkAction.st
```iecst
(** 2021-08-01 **)
ACTION Act_LinkAction:

	IF p_bLinkStartupRun = TRUE THEN
		p_eAct ACCESS p_StartupUSHermesAAct;
	ELSE
		p_eAct ACCESS ADR(eAct);

		IF EDGEPOS(p_eLinkMcParamUSCommMod = McSetCommModHermes) THEN
			bHermesRun	:= TRUE;
			bHermesStop	:= FALSE;
		END_IF

		IF EDGENEG(p_eLinkMcParamUSCommMod = McSetCommModHermes) THEN
			bHermesRun	:= FALSE;
			bHermesStop	:= TRUE;
		END_IF

		IF bHermesRun = TRUE THEN
			p_eAct	:= HermesActBGStartRun;

			IF (eStat = HermesActBGStartRun) AND (eStatus = Done) THEN
				p_eAct		:= HermesActIdle;
				bHermesRun	:= FALSE;
			END_IF
		END_IF

		IF bHermesStop = TRUE THEN
			p_eAct	:= HermesActBGStopRun;

			IF (eStat = HermesActBGStopRun) AND (eStatus = Done) THEN
				p_eAct		:= HermesActIdle;
				bHermesStop	:= FALSE;
			END_IF
		END_IF

		fbDlyTmr(IN := TRUE);
		IF fbDlyTmr.Q THEN
			fbDeleteLogTmr (IN := TRUE);
			IF fbDeleteLogTmr.Q AND eStatus <> Busy THEN
				p_eAct := HermesActDeleteOldLog;
				IF eStat = HermesActDeleteOldLog AND eStatus = Done THEN
					p_eAct := HermesActIdle;
					fbDlyTmr (IN := FALSE);
					fbDeleteLogTmr (IN := FALSE);
				END_IF
			END_IF
		END_IF

	END_IF

END_ACTION
```

#### Act_Main.st
```iecst
(** 2021-08-01 **)
ACTION Act_Main:

	IF eStatOld <> eStat THEN
		fbFileOldDel1(bEn := FALSE);

		sStatTxt	:= a_sStatText[eStat];

		eStatOld	:= eStat;

		eStatus		:= Busy;
	END_IF

	//Main
	CASE eStat OF

		HermesActIdle:
			eStatus	:= Idle;

		HermesActBGStartRun:
			IF eStatus = Idle OR eStatus = Busy THEN

				bRun	:= TRUE;
				bStop	:= FALSE;
				eStatus	:= Done;

			END_IF

		HermesActBGStopRun:
			IF eStatus = Idle OR eStatus = Busy THEN

				bStop	:= TRUE;
				eStatus	:= Done;

			END_IF

		HermesActDeleteOldLog:
			IF eStatus = Idle OR eStatus = Busy THEN

				eStatus	:= Busy;

				fbFileOldDel1.dtDTNow	:= p_dtCurrDT;
				fbFileOldDel1(bEn := TRUE);
				IF fbFileOldDel1.udiStatus = 0 THEN
					eStatus	:= Done;
				ELSIF fbFileOldDel1.udiStatus < 65534 THEN
					eStatus		:= Error;

					IF fbFileOldDel1.udiStatus = 1910 THEN
						udiStatus	:= 10154;	//Get Directory Info Error While Deleting Old Log
					ELSIF fbFileOldDel1.udiStatus = 1911 THEN
						udiStatus	:= 10155;	//Directory Read Error While Deleting Old Log
					ELSIF fbFileOldDel1.udiStatus = 1912 THEN
						udiStatus	:= 10156;	//File Delete Error While Deleting Old Log
					ELSE
						udiStatus	:= fbFileOldDel1.udiStatus;
					END_IF
				END_IF

			END_IF

		ELSE
			IF eStatus = Idle OR eStatus = Busy THEN
				eStatus	:= Done;
			END_IF

	END_CASE

END_ACTION
```

#### Act_Main_Disable.st
```iecst
(** 2021-08-01 **)
ACTION Act_Main_Disable:

	bConnected		:= FALSE;
	bHandshakeDone	:= FALSE;
	bAccDataReq		:= FALSE;
	bOverWriteSlt	:= FALSE;
	bOverWriteWidth	:= FALSE;
	bUSRdy			:= FALSE;
	bDSRdy			:= FALSE;
	bTransporting	:= FALSE;
	bStopTransport	:= FALSE;

END_ACTION
```

#### Init.st
```iecst
(** 2021-08-01 **)
PROGRAM _INIT

	(* Always Change If Project Change *)

	//Pass Address To Global Address For External Use
	//Action, State & Status
	p_USHermesAStat		:= ADR(eStat);
	p_USHermesAStatus	:= ADR(eMainStatus);
	p_USHermesAStatTxt	:= ADR(sStatTxt);

	//Alarm
	p_USHermesAAlmData	:= ADR(tyAlmData);
	p_USHermesAAlmData1	:= ADR(tyAlmData1);
	p_USHermesAAlmData2	:= ADR(tyAlmData2);
	p_USHermesAAlmData3	:= ADR(tyAlmData3);
	p_USHermesAAlmData4	:= ADR(tyAlmData4);
	p_USHermesAAlmData5	:= ADR(tyAlmData5);
	p_USHermesAInfoData	:= ADR(tyInfoData);
	p_USHermesAInfoData1	:= ADR(tyInfoData1);
	p_USHermesAInfoData2	:= ADR(tyInfoData2);

	//Output
	p_USHermesATableDataBrdAvl		:= ADR(a_tyXMLTableDataBrdAvl);
	p_USHermesATableDataBrdAvlTtlIdx	:= ADR(iXMLTableDataBrdAvlTtlIdx);
	p_USHermesAConnected				:= ADR(bConnected);
	p_USHermesAHandshakeDone			:= ADR(bHandshakeDone);
	p_USHermesAAccDataReq			:= ADR(bAccDataReq);
	p_USHermesABFAccDataReq			:= ADR(bBFAccDataReq);
	p_USHermesAOverWriteSlt			:= ADR(bOverWriteSlt);
	p_USHermesAOverWriteWidth		:= ADR(bOverWriteWidth);
	p_USHermesAReqRecipeNm			:= ADR(sReqRecipeNm);
	p_USHermesAReqWidthInUM			:= ADR(diReqWidthInUM);
	p_USHermesAReqMinSltValue		:= ADR(diReqMinSltValue);
	p_USHermesAReqMaxSltValue		:= ADR(diReqMaxSltValue);
	p_USHermesAReqPitch				:= ADR(diReqPitch);
	p_USHermesAUSRdy					:= ADR(bUSRdy);
	p_USHermesADSRdy					:= ADR(bDSRdy);
	p_USHermesAUSGdRdy				:= ADR(bUSGdRdy);
	p_USHermesADSGdRdy				:= ADR(bDSGdRdy);
	p_USHermesATransporting			:= ADR(bTransporting);
	p_USHermesAStopTransport			:= ADR(bStopTransport);
	p_USHermesABlkUS					:= ADR(bBlkUS);
	p_USHermesAInternalSnd			:= ADR(sInternalSnd);
	p_USHermesAAccDataMnl			:= ADR(bAccDataMnl);
	p_USHermesAStopTransportSnd		:= ADR(bStopTransportSnd); //bStopTransportSnd for SupervisoryHermes "BoardArrived"
	p_USHermesABoardArrivedData      := ADR(tyBoardArrivedInfo); //"BoardArrived" data for SupervisoryHermes
	p_USHermesARcvBoardInfoOk        := ADR(bRcvBoardInfoOk);
	p_USHermesARcvbBoardInfoIncompl  := ADR(bRcvBoardInfoIncompl);
	p_USHermesABoardInfoData         := ADR(tySendBoardInfoAcc); //Pass "SendBoardInfo" data for DSHermes "BoardAvailable", for inserted PCB
	p_USHermesANextAvlPCBTimer       := ADR(tNextPCBTm); //Time available for Next PCB from B.F, use this to make decisionto get board from which upstream if there are multiple several upstream
	p_USHermesAManuallInsertLastZone := ADR(bManuallInsertLastZone); //used to block board transfer to last zone to allow operator insert PCB back to last zone
	p_USHermesABoardAvailableRcv           := ADR (tyBoardAvailableRcv);   // Pass Receive data to Supervisory
	p_USHermesABoardForecastRcv            := ADR  (tyBoardForecastAcc);   // Pass Receive data to Supervisory

	//for AutoRcp
	p_USHermesABAAccepted :=  ADR(bBaReceivedInRdyState);
	p_USHermesABFAccepted :=  ADR(bBfReceivedInRdyState);
//	p_USHermesABfRcvInRdyState := ADR(bBfReceivedInRdyState);
//	p_USHermesABaRcvInRdyState := ADR(bBaReceivedInRdyState);
	//for Opcon
	p_USHermesATopBtmBarcode			:= ADR(sTopBtmBarcode);

	(* Always Change If Project Change *)
END_PROGRAM
```

### USHermesB.var - Change By Project
```iecst
(*2019-06-10*)
(**)
(*Action & State & Status*)
VAR
	p_USHermesBStat : UDINT;
	p_USHermesBStatus : UDINT;
	p_USHermesBStatTxt : UDINT;
END_VAR
(**)
(*Alarm*)
VAR
	p_USHermesBAlmData : UDINT;
	p_USHermesBAlmData1 : UDINT;
	p_USHermesBAlmData2 : UDINT;
	p_USHermesBAlmData3 : UDINT;
	p_USHermesBAlmData4 : UDINT;
	p_USHermesBAlmData5 : UDINT;
	p_USHermesBInfoData : UDINT;
	p_USHermesBInfoData1 : UDINT;
	p_USHermesBInfoData2 : UDINT;
END_VAR
(**)
(*Output*)
VAR
	p_USHermesBTableDataBrdAvl : UDINT;
	p_USHermesBTableDataBrdAvlTtlIdx : UDINT;
	p_USHermesBConnected : UDINT;
	p_USHermesBHandshakeDone : UDINT;
	p_USHermesBAccDataReq : UDINT;
	p_USHermesBBFAccDataReq : UDINT;
	p_USHermesBOverWriteSlt : UDINT;
	p_USHermesBOverWriteWidth : UDINT;
	p_USHermesBReqRecipeNm : UDINT;
	p_USHermesBReqWidthInUM : UDINT;
	p_USHermesBReqMinSltValue : UDINT;
	p_USHermesBReqMaxSltValue : UDINT;
	p_USHermesBReqPitch : UDINT;
	p_USHermesBUSRdy : UDINT;
	p_USHermesBDSRdy : UDINT;
	p_USHermesBUSGdRdy : UDINT;
	p_USHermesBDSGdRdy : UDINT;
	p_USHermesBTransporting : UDINT;
	p_USHermesBStopTransport : UDINT;
	p_USHermesBBlkUS : UDINT;
	p_USHermesBInternalSnd : UDINT;
	p_USHermesBAccDataMnl : UDINT;
	p_USHermesBStopTransportSnd : UDINT;
	p_USHermesBBoardArrivedData : UDINT;
	p_USHermesBRcvBoardInfoOk : UDINT;
	p_USHermesBRcvbBoardInfoIncompl : UDINT;
	p_USHermesBBoardInfoData : UDINT;
	p_USHermesBNextAvlPCBTimer : UDINT;
	p_USHermesBManuallInsertLastZone : UDINT;
	p_USHermesBBoardAvailableRcv : UDINT;
	p_USHermesBBoardForecastRcv : UDINT;
END_VAR
(*Changed*)
VAR
	p_USHermesBBAAccepted : UDINT;
	p_USHermesBBFAccepted : UDINT;
END_VAR
```

### Program Logical/Hermes/USHermesB (IEC, version 1.00.0) - 1.00.0 - NtHermes v5.00.0 , NtTCP v5.00.0 , NtMessage v5.00.0

#### Init.st - Change By Project
```iecst
(** 2021-08-01 **)
PROGRAM _INIT

	(* Always Change If Project Change *)

	//Pass Address To Global Address For External Use
	//Action, State & Status
	p_USHermesBStat		:= ADR(eStat);
	p_USHermesBStatus	:= ADR(eMainStatus);
	p_USHermesBStatTxt	:= ADR(sStatTxt);

	//Alarm
	p_USHermesBAlmData	:= ADR(tyAlmData);
	p_USHermesBAlmData1	:= ADR(tyAlmData1);
	p_USHermesBAlmData2	:= ADR(tyAlmData2);
	p_USHermesBAlmData3	:= ADR(tyAlmData3);
	p_USHermesBAlmData4	:= ADR(tyAlmData4);
	p_USHermesBAlmData5	:= ADR(tyAlmData5);
	p_USHermesBInfoData	:= ADR(tyInfoData);
	p_USHermesBInfoData1	:= ADR(tyInfoData1);
	p_USHermesBInfoData2	:= ADR(tyInfoData2);

	//Output
	p_USHermesBTableDataBrdAvl		:= ADR(a_tyXMLTableDataBrdAvl);
	p_USHermesBTableDataBrdAvlTtlIdx	:= ADR(iXMLTableDataBrdAvlTtlIdx);
	p_USHermesBConnected				:= ADR(bConnected);
	p_USHermesBHandshakeDone			:= ADR(bHandshakeDone);
	p_USHermesBAccDataReq			:= ADR(bAccDataReq);
	p_USHermesBBFAccDataReq			:= ADR(bBFAccDataReq);
	p_USHermesBOverWriteSlt			:= ADR(bOverWriteSlt);
	p_USHermesBOverWriteWidth		:= ADR(bOverWriteWidth);
	p_USHermesBReqRecipeNm			:= ADR(sReqRecipeNm);
	p_USHermesBReqWidthInUM			:= ADR(diReqWidthInUM);
	p_USHermesBReqMinSltValue		:= ADR(diReqMinSltValue);
	p_USHermesBReqMaxSltValue		:= ADR(diReqMaxSltValue);
	p_USHermesBReqPitch				:= ADR(diReqPitch);
	p_USHermesBUSRdy					:= ADR(bUSRdy);
	p_USHermesBDSRdy					:= ADR(bDSRdy);
	p_USHermesBUSGdRdy				:= ADR(bUSGdRdy);
	p_USHermesBDSGdRdy				:= ADR(bDSGdRdy);
	p_USHermesBTransporting			:= ADR(bTransporting);
	p_USHermesBStopTransport			:= ADR(bStopTransport);
	p_USHermesBBlkUS					:= ADR(bBlkUS);
	p_USHermesBInternalSnd			:= ADR(sInternalSnd);
	p_USHermesBAccDataMnl			:= ADR(bAccDataMnl);
	p_USHermesBStopTransportSnd		:= ADR(bStopTransportSnd); //bStopTransportSnd for SupervisoryHermes "BoardArrived"
	p_USHermesBBoardArrivedData      := ADR(tyBoardArrivedInfo); //"BoardArrived" data for SupervisoryHermes
	p_USHermesBRcvBoardInfoOk        := ADR(bRcvBoardInfoOk);
	p_USHermesBRcvbBoardInfoIncompl  := ADR(bRcvBoardInfoIncompl);
	p_USHermesBBoardInfoData         := ADR(tySendBoardInfoAcc); //Pass "SendBoardInfo" data for DSHermes "BoardAvailable", for inserted PCB
	p_USHermesBNextAvlPCBTimer       := ADR(tNextPCBTm); //Time available for Next PCB from B.F, use this to make decisionto get board from which upstream if there are multiple several upstream
	p_USHermesBManuallInsertLastZone := ADR(bManuallInsertLastZone); //used to block board transfer to last zone to allow operator insert PCB back to last zone
	p_USHermesBBoardAvailableRcv           := ADR (tyBoardAvailableRcv);   // Pass Receive data to Supervisory
	p_USHermesBBoardForecastRcv            := ADR  (tyBoardForecastAcc);   // Pass Receive data to Supervisory

	//for AutoRcp
	p_USHermesBBAAccepted :=  ADR(bBaReceivedInRdyState);
	p_USHermesBBFAccepted :=  ADR(bBfReceivedInRdyState);

	(* Always Change If Project Change *)
END_PROGRAM
```

#### Act_InitGlobal.st - Change By Project
```iecst
(** 2021-08-01 **)
ACTION Act_InitGlobal:

	(* Always Change If Project Change *)

	//Pass Data To Link
	p_bLinkStartupRun ACCESS p_StartupRun;
	p_eLinkMcParamUSCommMod ACCESS p_McParamUSCommBMod;
	p_bLinkNtParamProjLaneBPrep ACCESS p_NtParamProjLaneBPrep;
	//p_eLinkConvDir ACCESS p_NtParamProjConvDir;
	p_bLinkDILeftSen ACCESS p_DIConvLftSen;
	//p_bLinkDIRightSen ACCESS p_DIConvRgtSen;

	p_eLinkTravLifULPosGo ACCESS p_OpsTravLifULPosGo;
	p_bLinkOpsTravLifULUSComm ACCESS p_OpsTravLifULUSComm;

//	p_bLinkOpsGConv1HvBrd ACCESS p_ConvHvBrd;
//	p_bLinkOpsGConv2HvBrd ACCESS p_OpsGConv2HvBrd; //Zone 2 and so on.
//	p_bLinkOpsGConv1StepChkInitDone ACCESS p_OpsConvStepChkInit;
//	p_bLinkOpsGConv2StepChkInitDone ACCESS p_OpsGConv2StepChkInitDone;  //Zone 2 and so on.
//	p_bLinkDIPresentSen ACCESS p_DIBrdStackPresentSen;

	//Pass Data To Internal Use
	p_udiRstErr ACCESS p_RstErrReset;
	p_bPrep ACCESS p_NtParamHermesPrep;
	p_tyParam ACCESS p_HermesUSParam1;
	p_sIPAddr ACCESS p_HWInfoIPAddr;
	p_tyDTStructure ACCESS p_TimeCurrDTStruct;
	p_dtCurrDT ACCESS p_TimeCurrDT;
	p_sMcId ACCESS p_McParamMcNm;
	p_sRecipeNm ACCESS p_ProdRcpCurrRcp0Nm;
	p_diWidthInUM ACCESS p_ProdRcpCurrRcp0Width;
	p_udiAliveIdleTimeInSec ACCESS p_NtParamUSHermesAAliveTmInSec;
	p_tConnTimeOut ACCESS p_NtParamUSHermesAConnTO;
	p_diTransferInTO ACCESS p_McParamTranInErrDlyTm;
	p_bInterruptSen ACCESS p_DIConvLftSen;
	p_bOpsRun ACCESS p_OpsRun;
	p_udiFileKeepDay ACCESS p_NtParamUSHermesAFileKeepDay;
	p_sProgNm ACCESS p_NtParamUSHermesAProgNm;
	p_bNtSettingsLoadDone ACCESS p_StartupNtSettingsLoadDone;
//	p_bAccDataRdy ACCESS p_USHermesUSRdy;
	p_bRmtPrep ACCESS p_NtParamHermesRmtPrep;
	p_bRmtEn ACCESS p_McParamHermesRmtEn;
	p_bSvyPrep ACCESS p_NtParamHermesSvyPrep;
	p_bSvyEn ACCESS p_McParamHermesSvyEn;
	pa_tyProdRcpList ACCESS p_ProdRcpCurrList;
	p_tyProdRcpCurrRcp ACCESS p_ProdRcpCurrRcp0;
	p_bMcParamMnlAccData ACCESS p_McParamMnlAccDat;
	p_bOpsGConv1HvBrd ACCESS p_PshrConvHvBrd;//p_ConvHvBrd; //Take Zone 1's Have Board
	//p_bManualInsertZoneHvBrd ACCESS p_ConvHvBrd; //Take Manual Insesrt Zone's Have Board
	//p_bManualInsertEndSen ACCESS p_DIConvRgtSen; //Manual insert sensor position, for example exit sensor of attached output conveyor, or Last Zone conveyor exit sensor
	p_bUIAccData ACCESS p_UIProdAccData;
	p_bQueryBoardInfo ACCESS p_UIQueryBoardInfo;
	p_sTopBarcode ACCESS p_UITravLifTopBarcode;
	p_sBottomBarcode ACCESS p_UITravLifBottomBarcode;
	p_tyHermesConfiguration ACCESS p_HermesConfiguration;
	//p_bTransportFinished ACCESS p_DSHermesTransportFinishedSnd; //used to reset bManuallInsertLastZone

	p_bSiemensMcModeChgPrep ACCESS p_McParamSiemensPrep;          //ADD   Include ReplyWorkOrderID & Machine mode changeover
	p_usiLinkProdRcpCurrRcpMcMod ACCESS p_ProdRcpCurrRcp0McMod;      //Add
	p_bNewIncomingBoard ACCESS p_NewIncomingBoard;
	p_bQueryBypassWorkOrder ACCESS p_QueryBypassWorkOrder;

	p_bNtParamAutoRcpPrep ACCESS p_NtParamAutoRcpPrep;
	p_bMcParamAutoRcpDis  ACCESS p_McParamAutoRcpDisable;
	p_eNtParamAutoRcpPrecededBy ACCESS p_NtParamAutoRcpPrecededBy;
	(* Always Change If Project Change *)
END_ACTION
```
